// TIA Portal V19 export
FUNCTION_BLOCK "A0303_Manager_FB"   // FB14, LAD
// stored: MemoryReserve 100, SetENOAutomatically false
   VAR_INPUT
      AreaInterface : "AreaInterface";
      DataIn : Struct
         LsCheckPassaggio_Coda : Bool;   // FTC LETTURA STRATO DEPOSITATO TESTA
         LsCheckPassaggio_Testa : Bool;   // FTC LETTURA STRATO DEPOSITATO TESTA
         LsPezzoPosMax_Coda : Bool;
         LsPezzoPosMax_Testa : Bool;
         SemiAut_Pb : Bool;
      END_STRUCT;
      CIn : Struct
         PareggiatoreTesta : Struct
            Ax : "Positioning_DOL_Machine_COut";
         END_STRUCT;
         PareggiatoreCoda : Struct
            Ax : "Positioning_DOL_Machine_COut";
         END_STRUCT;
         Spalle : Struct
            Testa : Struct
               Ax : "Positioning_DOL_Machine_COut";
            END_STRUCT;
            Coda : Struct
               Ax : "Positioning_DOL_Machine_COut";
            END_STRUCT;
         END_STRUCT;
         Spintore : Struct
            Vrt : "ValveMachine_COut";
            Orz : "ValveMachine_COut";
         END_STRUCT;
         TraslazioneStrato : Struct
            Ax_Testa : "Positioning_EPOS_Machine_COut";
            Ax_Coda : "Positioning_EPOS_Machine_COut";
            Manip_Sostegno : "ValveMachine_COut";
            Manip_Pareggiatore : "ValveMachine_COut";
            SostegnoVrt : "ValveMachine_COut";
            IsMeasuring : Bool;
         END_STRUCT;
         Sollevamento : Struct
            Ax_Testa : "Positioning_DOL_Machine_COut";
            Ax_Coda : "Positioning_DOL_Machine_COut";
         END_STRUCT;
         Sostegno : Struct
            Testa : Struct
               Ax : "Positioning_DOL_Machine_COut";
               Paletto : Struct
                  CtrlSafe : Bool;
                  Standstill : Bool;
                  Rest_CheckNext : Bool;
                  Work_CheckNext : Bool;
                  Pos : Int;
                  RestPosition : Bool;
               END_STRUCT;
            END_STRUCT;
            Coda : Struct
               Ax : "Positioning_DOL_Machine_COut";
               Paletto : Struct
                  CtrlSafe : Bool;
                  Standstill : Bool;
                  Rest_CheckNext : Bool;
                  Work_CheckNext : Bool;
                  Pos : Int;
                  RestPosition : Bool;
               END_STRUCT;
            END_STRUCT;
         END_STRUCT;
         Navetta : Struct
            ReadyToRecive : Bool;
            OutOfWorkspace : Bool;
            InPosizioneDiDeposito : Bool;
            InPosizioneDiPrelievo : Bool;
            InPosizioneDiPrePrelievo : Bool;
            RequestDeposito : Bool;
            RequestPrelievo : Bool;
         END_STRUCT;
         ProdManager : "Prod_Beam_Ctrl";
      END_STRUCT;
   END_VAR
   VAR_OUTPUT
      MachineInterface : "MachineInterface";
      COut : Struct
         Spalla : Struct
            Testa : "Positioning_DOL_Machine_Manager";
            Coda : "Positioning_DOL_Machine_Manager";
         END_STRUCT;
         Spintore : Struct
            EnableStopDoorOpeningReq : Bool;
            EnableStopInPhase : Bool;
            EnableStopProgrammed : Bool;
            Control_ON : Bool;
            CanMoveFreely : Bool;
            Rest : Bool;
            Work : Bool;
         END_STRUCT;
         Trasporto : Struct
            EnableStopDoorOpeningReq : Bool;
            EnableStopInPhase : Bool;
            EnableStopProgrammed : Bool;
            Control_ON : Bool;
            CanMoveFreely : Bool;
            OP : Struct
               VAI_A_PRELIEVO : Bool;
               PRELIEVO : Bool;
               VAI_A_DEPOSITO : Bool;
               DEPOSITO : Bool;
            END_STRUCT;
         END_STRUCT;
         Sollevatore : Struct
            EnableStopDoorOpeningReq : Bool;
            EnableStopInPhase : Bool;
            EnableStopProgrammed : Bool;
            Control_ON : Bool;
            CanMoveFreely : Bool;
            TargetPosition : LReal;
            OP : Struct
               PRELIEVO : Bool;
               PRE_DEPOSITO : Bool;
               DEPOSITO : Bool;
            END_STRUCT;
         END_STRUCT;
         Sostegno : Struct
            Testa : Struct
               EnableStopDoorOpeningReq : Bool;
               EnableStopInPhase : Bool;
               EnableStopProgrammed : Bool;
               Control_ON : Bool;
               CanMoveFreely : Bool;
               Phase : Struct
                  VAI_A_LAVORO : Bool;
                  VAI_A_RIPOSO : Bool;
               END_STRUCT;
               Ax : Struct
                  Pos { ExternalVisible := 'False'; ExternalWritable := 'False'} : LReal;
               END_STRUCT;
               Paletti : Struct
                  PosPaletto : Int;
                  Pos1Collision : Bool;
                  Pos2Collision : Bool;
               END_STRUCT;
            END_STRUCT;
            Coda : Struct
               EnableStopDoorOpeningReq : Bool;
               EnableStopInPhase : Bool;
               EnableStopProgrammed : Bool;
               Control_ON : Bool;
               CanMoveFreely : Bool;
               Phase : Struct
                  VAI_A_LAVORO : Bool;
                  VAI_A_RIPOSO : Bool;
               END_STRUCT;
               Ax : Struct
                  Pos { ExternalVisible := 'False'; ExternalWritable := 'False'} : LReal;
               END_STRUCT;
               Paletti : Struct
                  PosPaletto : Int;
                  Pos1Collision : Bool;
                  Pos2Collision : Bool;
               END_STRUCT;
            END_STRUCT;
         END_STRUCT;
         Manipolatore : Struct
            ReadyToRecive : Bool;
         END_STRUCT;
      END_STRUCT;
   END_VAR
   VAR_IN_OUT
      Par : Struct
         Antiribaltamento : Struct
            Offset_Pos : LReal;
         END_STRUCT;
      END_STRUCT;
      Par_Trasporto : Struct
         PosPrelievo : LReal;
         PosDeposito : LReal;
         ToleranceWindow : LReal;
      END_STRUCT;
      Par_Sollevatore : Struct
         PosDeposito : LReal;
         OffsetPrelievo : LReal;
         ToleranceWindow : LReal;
      END_STRUCT;
      Par_SostegnoAntirib : Struct
         RestPosition : LReal;
         ToleranceWindow : LReal;
         PosTimeout : Time;
      END_STRUCT;
      Par_Spalla_Testa : Struct
         MinDistanzaConParegg : LReal;
         ToleranceWindow : LReal;
      END_STRUCT;
      Par_Spalla_Coda : Struct
         MinDistanzaConParegg : LReal;
         ToleranceWindow : LReal;
      END_STRUCT;
   END_VAR
   VAR
      Alarm : Struct
         TrkPassaggioPezzo : Bool;
         TrkPreparationAlreadyFull : Bool;
         TrkStackerAlreadyFull : Bool;
         PaccoOltreLimiteMax : Bool;
         STOP_FineTurno : Bool;
         STOP_End_Of_Proroduction : Bool;
         STOP_ControlloQualita : Bool;
         STOP_Inattività : Bool;
      END_STRUCT;
      Warning : Struct
         IsWaiting_NoPiecesBefore : Bool;
         IsWaiting_NoPiecesBefore_A01NotInCycle : Bool;
         IsWaiting_NoPiecesBefore_A02NotInCycle : Bool;
         IsWaiting_NoPiecesBefore_A03NotInCycle : Bool;
         IsWaiting_ShuttleUnload : Bool;
         IsWaiting_PezziDaRintegrare : Bool;
         STOP_End_Of_Proroduction : Bool;
         STOP_FineTurno : Bool;
         STOP_ControlloQualita : Bool;
         MissingCnd : Struct
            SollevatoreNotReadyToRecive : Bool;
         END_STRUCT;
      END_STRUCT;
      OP_CND : Struct
         Trasporto : Struct
            VaiAPrelievo : Array[0..15] of "OpCnd";
            Prelievo { S7_SetPoint := 'True'} : Array[0..15] of "OpCnd";
            VaiADeposito : Array[0..15] of "OpCnd";
            Deposito : Array[0..15] of "OpCnd";
         END_STRUCT;
      END_STRUCT;
      Ctrl : Struct
         Stop : Bool;
         Cycle : Struct
            Trasferimento : Struct
               VaiAPrelievo : Bool;   // CICLO - Vai a Posizione di prelievo
               Prelievo : Bool;   // CICLO - Prelievo
               VaiADeposito : Bool;   // CICLO - Vai a Posizione di deposito
               Deposito : Bool;   // CICLO - Deposito
            END_STRUCT;
            Sollevamento : Struct
               Prelievo : Bool;
               Deposito : Bool;
               PreDeposito : Bool;
            END_STRUCT;
            SostegnoAntirib_Testa : Struct
               VaiALavoro : Bool;
               VaiARiposo : Bool;
               CyclePos : LReal;
               PalettoPos : Int;
            END_STRUCT;
            SostegnoAntirib_Coda : Struct
               VaiALavoro : Bool;
               VaiARiposo : Bool;
               CyclePos : LReal;
               PalettoPos : Int;
            END_STRUCT;
         END_STRUCT;
         BTrk : Struct
            B3ToLayer1 : Bool;
            TransferToStacker : Bool;
         END_STRUCT;
         Spintore : Struct
            Vrt : Struct
               Rest : Bool;
               Work : Bool;
            END_STRUCT;
            Orz : Struct
               Rest : Bool;
               Work : Bool;
            END_STRUCT;
            Work : Bool;
            Rest : Bool;
         END_STRUCT;
         Spalle : Struct
            Testa : Struct
               MoveToPos : Bool;
               Pos : LReal;
            END_STRUCT;
            Coda : Struct
               MoveToPos : Bool;
               Pos : LReal;
            END_STRUCT;
         END_STRUCT;
         TraslazioneStrato : Struct
            Ax : Struct
               MovePrelievo : Bool;
               MoveDeposito : Bool;
               PosDeposito : LReal;
               PosPrelievo : LReal;
            END_STRUCT;
            SostegnoVrt : Struct
               Rest : Bool;
               Work : Bool;
            END_STRUCT;
            Manip_Sostegno : Struct
               Rest : Bool;
               Work : Bool;
            END_STRUCT;
            Manip_Pareggiatore : Struct
               Rest : Bool;
               Work : Bool;
            END_STRUCT;
         END_STRUCT;
      END_STRUCT;
      Sts : Struct
         AlarmsPresence : Bool;
         WarningsPresence : Bool;
         IsStandstill : Bool;
         SemiAut : Struct
            ON : Bool;
            PbMaterialFwd : Bool;
            Request : Bool;
         END_STRUCT;
         SpallaTesta : Struct
            InCyclePos : Bool;
         END_STRUCT;
         SpallaCoda : Struct
            InCyclePos : Bool;
         END_STRUCT;
         Sollevatore : Struct
            ReadyToRecive : Bool;
            InPrelievoPos : Bool;
            InPrePrelievoPos : Bool;
            InPosDeposito : Bool;
            InPosPreDeposito : Bool;
         END_STRUCT;
         Preparazione : Struct
            Completato : Bool;
         END_STRUCT;
         TraslazioneStrato : Struct
            InPosDeposito : Bool;
            InPosPrelievo : Bool;
            OutOfWorkspace : Bool;   // Fuori ingombro con sollevatore
            DropRequest : Bool;
         END_STRUCT;
         SostegnoTesta : Struct
            Ax : Struct
               InCyclePos : Bool;
               InRestPos : Bool;
            END_STRUCT;
            Paletto : Struct
               InCyclePos : Bool;
            END_STRUCT;
         END_STRUCT;
         SostegnoCoda : Struct
            Ax : Struct
               InCyclePos : Bool;
               InRestPos : Bool;
            END_STRUCT;
            Paletto : Struct
               InCyclePos : Bool;
            END_STRUCT;
         END_STRUCT;
         BTrk { ExternalAccessible := 'False'; ExternalVisible := 'False'; ExternalWritable := 'False'} : Struct
            ZonePreparationEmpty { S7_SetPoint := 'True'} : Bool;
            ZoneStackerEmpty : Bool;
            Actual_O_ID : DInt;
         END_STRUCT;
      END_STRUCT;
      AUX : Struct
         LsPosition1Coda_PE { ExternalAccessible := 'False'; ExternalVisible := 'False'; ExternalWritable := 'False'} : Bool;
         LsPosition1Coda_NE { ExternalAccessible := 'False'; ExternalVisible := 'False'; ExternalWritable := 'False'} : Bool;
         LsPosition1Testa_PE { ExternalAccessible := 'False'; ExternalVisible := 'False'; ExternalWritable := 'False'} : Bool;
         LsPosition1Testa_NE { ExternalAccessible := 'False'; ExternalVisible := 'False'; ExternalWritable := 'False'} : Bool;
         TrkToTransfer { ExternalAccessible := 'False'; ExternalVisible := 'False'; ExternalWritable := 'False'} : Bool;
         TrkToShuttle : Bool;
         SemiAut_Pb : Bool;
      END_STRUCT;
      TON_PassaggioPezzoAlarm : IEC_TIMER;
      TON_NoPiecesBefore : IEC_TIMER;
      TON_Stop { S7_SetPoint := 'True'} : IEC_TIMER;
      TON_StopPerInattivita { S7_SetPoint := 'True'} : IEC_TIMER;
      Attrezzamento : Struct
         Ready : Bool;
         FindNewID : Bool;
         RequestNewPosition : Bool;
         TargetSpalle : LReal;
         TargetSostegno : LReal;
         ID : DInt;
      END_STRUCT;
      CycleWithShortPiece : Bool;
      PE_Engaged_Coda : Bool;
      NE_Engaged_Coda : Bool;
      PE_Engaged_Testa : Bool;
      NE_Engaged_Testa : Bool;
      TON_CheckCompletato_Stacker : IEC_TIMER;
      TON_CheckCompletato_Preparation : IEC_TIMER;
   END_VAR
   VAR_TEMP
      PE : Struct
         LsPosition1_Coda : Bool;
         LsPosition1_Testa : Bool;
         TrkToTransfer : Bool;
         TrkToShuttle : Bool;
      END_STRUCT;
      NE : Struct
         LsPosition1_Coda : Bool;
         LsPosition1_Testa : Bool;
      END_STRUCT;
      BTrk_GetData : Struct   // BTrk letto dal MES
         indx : Int;   // Se trovato tra i TODO / ENDING / OUT questo è l'indice dove sono stati prelevati i dati
         Sts : Int;   // 0 = Non Trovato; 0 = ACT; 1 = TODO; 2=ENDING; 3 = OUT
         Item : "Prod_Item_small";
      END_STRUCT;
      BTrk_Absence : Bool;
      LayerTrk_Absence : Bool;
      O_ID_Precedenti : DInt;
      i : Int;
      EmptyNFound : Int;
      ShiftN : Int;
      TargetPrePositionSollevatore : LReal;
      TargetPositionSollevatore_Temp : LReal;
      TargetPositionSollevatore : LReal;
      TargetPreDepositoSollevatore : LReal;
      SollevatoreCodaInPrelievoPos : Bool;
      SollevatoreTestaInPrelievoPos : Bool;
      SollevatoreCodaInPrePrelievoPos : Bool;
      SollevatoreTestaInPrePrelievoPos : Bool;
      SollevatoreCodaInPosDeposito : Bool;
      SollevatoreTestaInPosDeposito : Bool;
      SollevatoreTestaInPosPreDeposito : Bool;
      SollevatoreCodaInPosPreDeposito : Bool;
      TrasportoTestaInPosDeposito : Bool;
      TrasportoTestaInPosPrelievo : Bool;
      TrasportoCodaInPosDeposito : Bool;
      TrasportoCodaInPosPrelievo : Bool;
      ShiftArrayOk : Int;
      TrkToStackerOk : Int;
      PieceToCheck_Presence : Bool;
      O_ID_Temp : DInt;
      ConteggioPezzi_Preparation : Int;
      ConteggioPezzi_Stacker : Int;
      ConteggioPezzi_Transfert : Int;
      MaxBeamsXLayer : Int;
      MaxLayer : Int;
   END_VAR
   VAR CONSTANT
      TrasportoOutOfWorkspace : LReal := -215.0;
   END_VAR
   VAR_TEMP   // added for the SCL form of the ladder/FBD networks
      _w1 : Bool;
      _w2 : Bool;
      _w3 : Bool;
      _w4 : Bool;
      _w5 : Bool;
   END_VAR
BEGIN

REGION Network 1 (SCL): Reset Alarms
   IF #AreaInterface.RstAlarms THEN
       #Alarm.TrkPassaggioPezzo := FALSE;
       #Alarm.TrkPreparationAlreadyFull := FALSE;
       #Alarm.TrkStackerAlreadyFull := FALSE;
       #Alarm.PaccoOltreLimiteMax := FALSE;
       #Alarm.STOP_End_Of_Proroduction := FALSE;
       #Alarm.STOP_FineTurno := FALSE;
       #Alarm.STOP_ControlloQualita := FALSE;
   END_IF;
END_REGION

REGION Network 2: Fronti Sensori
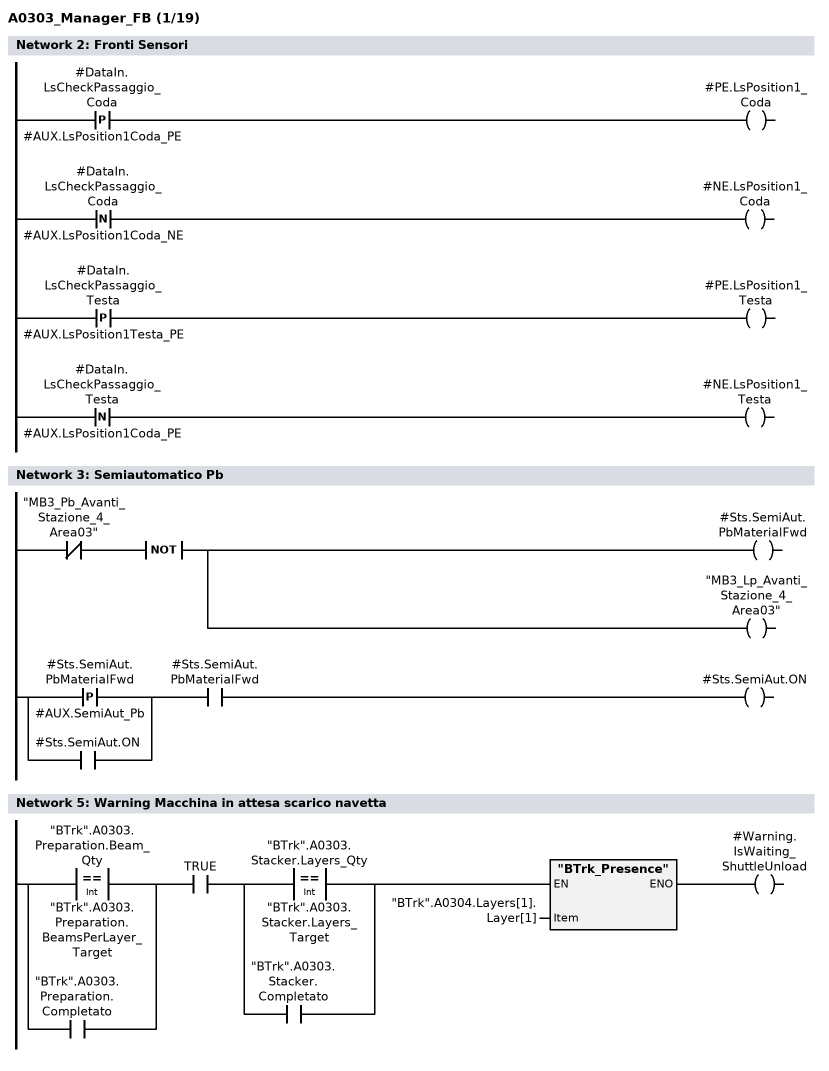
   RUNG wire#powerrail
      P_Contact(operand := #DataIn.LsCheckPassaggio_Coda, bit := #AUX.LsPosition1Coda_PE)
      Coil( #PE.LsPosition1_Coda )
   END_RUNG
   RUNG wire#powerrail
      N_Contact(operand := #DataIn.LsCheckPassaggio_Coda, bit := #AUX.LsPosition1Coda_NE)
      Coil( #NE.LsPosition1_Coda )
   END_RUNG
   RUNG wire#powerrail
      P_Contact(operand := #DataIn.LsCheckPassaggio_Testa, bit := #AUX.LsPosition1Testa_PE)
      Coil( #PE.LsPosition1_Testa )
   END_RUNG
   RUNG wire#powerrail
      N_Contact(operand := #DataIn.LsCheckPassaggio_Testa, bit := #AUX.LsPosition1Coda_PE)
      Coil( #NE.LsPosition1_Testa )
   END_RUNG
   // the same network as SCL:
   #_w1 := #DataIn.LsCheckPassaggio_Coda AND NOT #AUX.LsPosition1Coda_PE;   // rising edge of #DataIn.LsCheckPassaggio_Coda
   #AUX.LsPosition1Coda_PE := #DataIn.LsCheckPassaggio_Coda;
   #PE.LsPosition1_Coda := #_w1;
   #_w2 := NOT #DataIn.LsCheckPassaggio_Coda AND #AUX.LsPosition1Coda_NE;   // falling edge of #DataIn.LsCheckPassaggio_Coda
   #AUX.LsPosition1Coda_NE := #DataIn.LsCheckPassaggio_Coda;
   #NE.LsPosition1_Coda := #_w2;
   #_w3 := #DataIn.LsCheckPassaggio_Testa AND NOT #AUX.LsPosition1Testa_PE;   // rising edge of #DataIn.LsCheckPassaggio_Testa
   #AUX.LsPosition1Testa_PE := #DataIn.LsCheckPassaggio_Testa;
   #PE.LsPosition1_Testa := #_w3;
   #_w4 := NOT #DataIn.LsCheckPassaggio_Testa AND #AUX.LsPosition1Coda_PE;   // falling edge of #DataIn.LsCheckPassaggio_Testa
   #AUX.LsPosition1Coda_PE := #DataIn.LsCheckPassaggio_Testa;
   #NE.LsPosition1_Testa := #_w4;
END_REGION

REGION Network 3: Semiautomatico Pb
   RUNG wire#powerrail
      I_Contact( "MB3_Pb_Avanti_Stazione_4_Area03" )
      Not()
      wire#w1
      Coil( #Sts.SemiAut.PbMaterialFwd )
   END_RUNG
   RUNG wire#w1
      Coil( "MB3_Lp_Avanti_Stazione_4_Area03" )
   END_RUNG
   RUNG wire#powerrail
      P_Contact(operand := #Sts.SemiAut.PbMaterialFwd, bit := #AUX.SemiAut_Pb)
      wire#w2
      Contact( #Sts.SemiAut.PbMaterialFwd )
      Coil( #Sts.SemiAut.ON )
   END_RUNG
   RUNG wire#powerrail
      Contact( #Sts.SemiAut.ON )
   END_RUNG wire#w2
   // the same network as SCL:
   #Sts.SemiAut.PbMaterialFwd := NOT (NOT "MB3_Pb_Avanti_Stazione_4_Area03");
   "MB3_Lp_Avanti_Stazione_4_Area03" := NOT (NOT "MB3_Pb_Avanti_Stazione_4_Area03");
   #_w1 := #Sts.SemiAut.PbMaterialFwd AND NOT #AUX.SemiAut_Pb;   // rising edge of #Sts.SemiAut.PbMaterialFwd
   #AUX.SemiAut_Pb := #Sts.SemiAut.PbMaterialFwd;
   #Sts.SemiAut.ON := (#_w1 OR #Sts.SemiAut.ON) AND #Sts.SemiAut.PbMaterialFwd;
END_REGION

REGION Network 5: Warning Macchina in attesa scarico navetta
   RUNG wire#powerrail
      { S7_Templates := "SrcType := Int" } EQ_Contact(in1 := "BTrk".A0303.Preparation.Beam_Qty, in2 := "BTrk".A0303.Preparation.BeamsPerLayer_Target)
      wire#w1
      Contact( TRUE )
      wire#w2
      { S7_Templates := "SrcType := Int" } EQ_Contact(in1 := "BTrk".A0303.Stacker.Layers_Qty, in2 := "BTrk".A0303.Stacker.Layers_Target)
      wire#w3
      "BTrk_Presence"(Item := "BTrk".A0304.Layers[1].Layer[1])
      Coil( #Warning.IsWaiting_ShuttleUnload )
   END_RUNG
   RUNG wire#powerrail
      Contact( "BTrk".A0303.Preparation.Completato )
   END_RUNG wire#w1
   RUNG wire#w2
      Contact( "BTrk".A0303.Stacker.Completato )
   END_RUNG wire#w3
   // the same network as SCL:
   "BTrk_Presence"(EN := (("BTrk".A0303.Preparation.Beam_Qty = "BTrk".A0303.Preparation.BeamsPerLayer_Target) OR "BTrk".A0303.Preparation.Completato) AND TRUE AND (("BTrk".A0303.Stacker.Layers_Qty = "BTrk".A0303.Stacker.Layers_Target) OR "BTrk".A0303.Stacker.Completato),
                   Item := "BTrk".A0304.Layers[1].Layer[1],
                   ENO => #_w1);
   #Warning.IsWaiting_ShuttleUnload := #_w1;
END_REGION

REGION Network 6: Warning Macchina in attesa nessun pezzo in arrivo
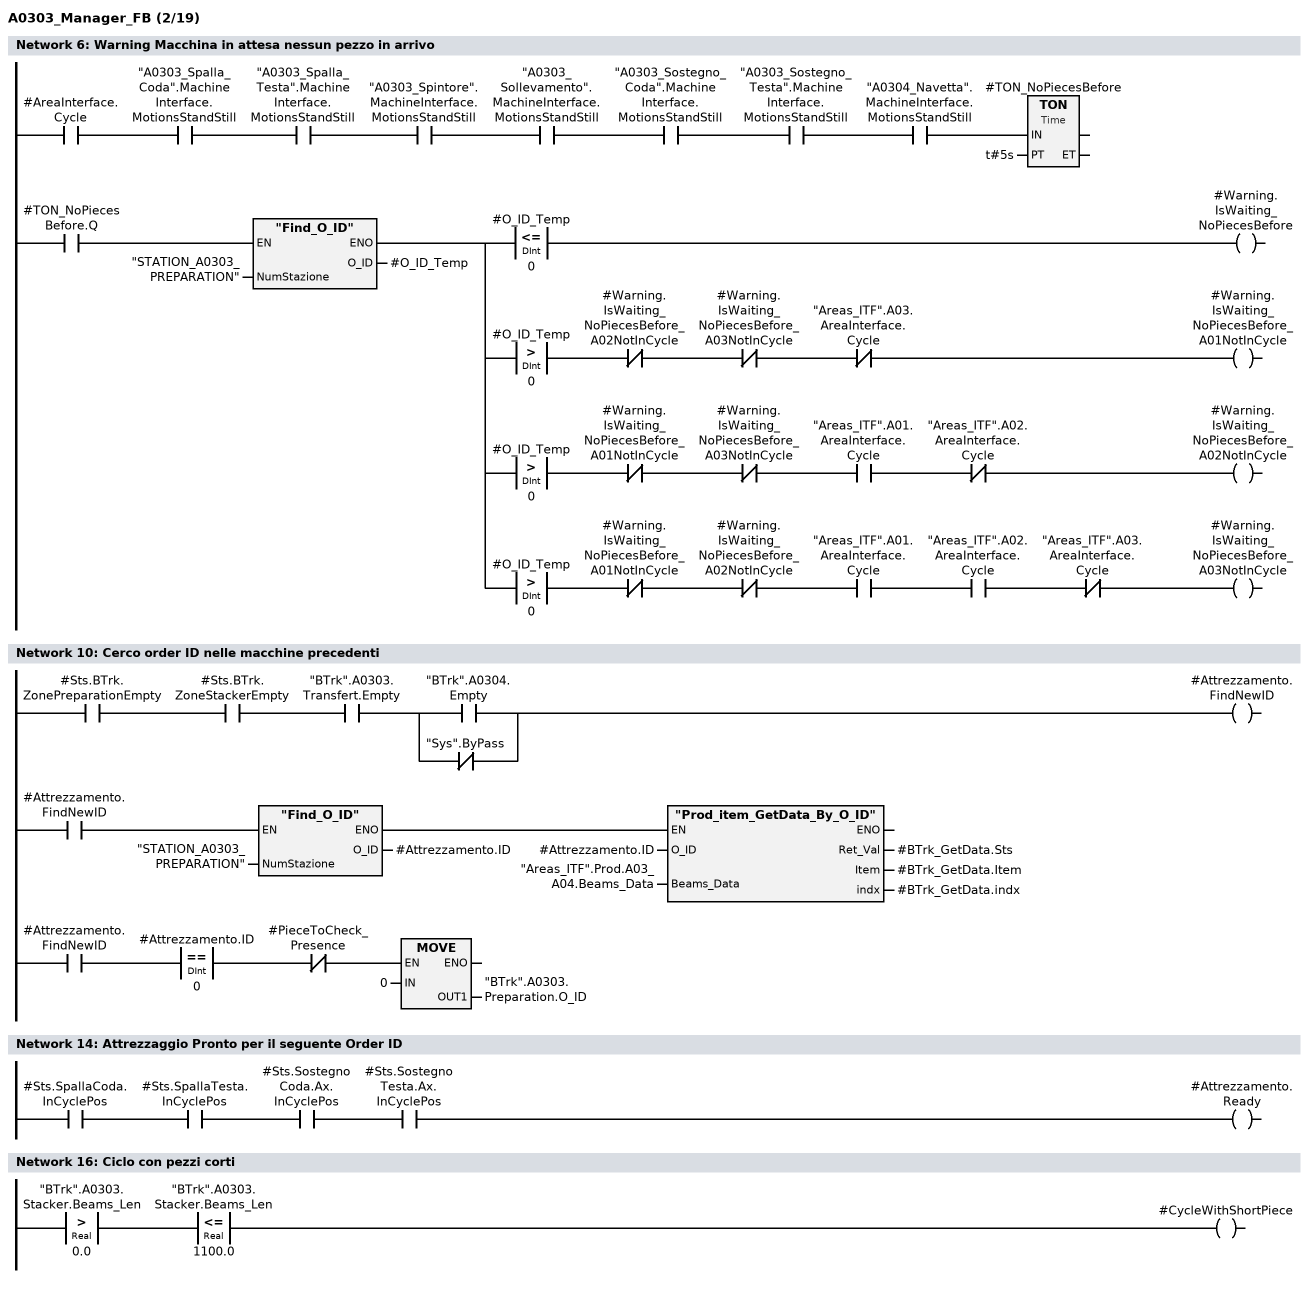
   RUNG wire#powerrail
      Contact( #AreaInterface.Cycle )
      Contact( "A0303_Spalla_Coda".MachineInterface.MotionsStandStill )
      Contact( "A0303_Spalla_Testa".MachineInterface.MotionsStandStill )
      Contact( "A0303_Spintore".MachineInterface.MotionsStandStill )
      Contact( "A0303_Sollevamento".MachineInterface.MotionsStandStill )
      Contact( "A0303_Sostegno_Coda".MachineInterface.MotionsStandStill )
      Contact( "A0303_Sostegno_Testa".MachineInterface.MotionsStandStill )
      Contact( "A0304_Navetta".MachineInterface.MotionsStandStill )
      { S7_Templates := "time_type := Time" } #TON_NoPiecesBefore.TON(pt := t#5s, et =>)
   END_RUNG
   RUNG wire#powerrail
      Contact( #TON_NoPiecesBefore.Q )
      "Find_O_ID"(NumStazione := "STATION_A0303_PREPARATION", O_ID => #O_ID_Temp)
      wire#w1
      { S7_Templates := "SrcType := DInt" } LE_Contact(in1 := #O_ID_Temp, in2 := 0)
      Coil( #Warning.IsWaiting_NoPiecesBefore )
   END_RUNG
   RUNG wire#w1
      { S7_Templates := "SrcType := DInt" } GT_Contact(in1 := #O_ID_Temp, in2 := 0)
      I_Contact( #Warning.IsWaiting_NoPiecesBefore_A02NotInCycle )
      I_Contact( #Warning.IsWaiting_NoPiecesBefore_A03NotInCycle )
      I_Contact( "Areas_ITF".A03.AreaInterface.Cycle )
      Coil( #Warning.IsWaiting_NoPiecesBefore_A01NotInCycle )
   END_RUNG
   RUNG wire#w1
      { S7_Templates := "SrcType := DInt" } GT_Contact(in1 := #O_ID_Temp, in2 := 0)
      I_Contact( #Warning.IsWaiting_NoPiecesBefore_A01NotInCycle )
      I_Contact( #Warning.IsWaiting_NoPiecesBefore_A03NotInCycle )
      Contact( "Areas_ITF".A01.AreaInterface.Cycle )
      I_Contact( "Areas_ITF".A02.AreaInterface.Cycle )
      Coil( #Warning.IsWaiting_NoPiecesBefore_A02NotInCycle )
   END_RUNG
   RUNG wire#w1
      { S7_Templates := "SrcType := DInt" } GT_Contact(in1 := #O_ID_Temp, in2 := 0)
      I_Contact( #Warning.IsWaiting_NoPiecesBefore_A01NotInCycle )
      I_Contact( #Warning.IsWaiting_NoPiecesBefore_A02NotInCycle )
      Contact( "Areas_ITF".A01.AreaInterface.Cycle )
      Contact( "Areas_ITF".A02.AreaInterface.Cycle )
      I_Contact( "Areas_ITF".A03.AreaInterface.Cycle )
      Coil( #Warning.IsWaiting_NoPiecesBefore_A03NotInCycle )
   END_RUNG
   // the same network as SCL:
   #TON_NoPiecesBefore.TON(IN := #AreaInterface.Cycle AND "A0303_Spalla_Coda".MachineInterface.MotionsStandStill AND "A0303_Spalla_Testa".MachineInterface.MotionsStandStill AND "A0303_Spintore".MachineInterface.MotionsStandStill AND "A0303_Sollevamento".MachineInterface.MotionsStandStill AND "A0303_Sostegno_Coda".MachineInterface.MotionsStandStill AND "A0303_Sostegno_Testa".MachineInterface.MotionsStandStill AND "A0304_Navetta".MachineInterface.MotionsStandStill,
                           PT := t#5s);
   "Find_O_ID"(EN := #TON_NoPiecesBefore.Q,
               NumStazione := "STATION_A0303_PREPARATION",
               O_ID => #O_ID_Temp,
               ENO => #_w1);
   #Warning.IsWaiting_NoPiecesBefore := #_w1 AND (#O_ID_Temp <= 0);
   #Warning.IsWaiting_NoPiecesBefore_A01NotInCycle := #_w1 AND (#O_ID_Temp > 0) AND NOT #Warning.IsWaiting_NoPiecesBefore_A02NotInCycle AND NOT #Warning.IsWaiting_NoPiecesBefore_A03NotInCycle AND NOT "Areas_ITF".A03.AreaInterface.Cycle;
   #Warning.IsWaiting_NoPiecesBefore_A02NotInCycle := #_w1 AND (#O_ID_Temp > 0) AND NOT #Warning.IsWaiting_NoPiecesBefore_A01NotInCycle AND NOT #Warning.IsWaiting_NoPiecesBefore_A03NotInCycle AND "Areas_ITF".A01.AreaInterface.Cycle AND NOT "Areas_ITF".A02.AreaInterface.Cycle;
   #Warning.IsWaiting_NoPiecesBefore_A03NotInCycle := #_w1 AND (#O_ID_Temp > 0) AND NOT #Warning.IsWaiting_NoPiecesBefore_A01NotInCycle AND NOT #Warning.IsWaiting_NoPiecesBefore_A02NotInCycle AND "Areas_ITF".A01.AreaInterface.Cycle AND "Areas_ITF".A02.AreaInterface.Cycle AND NOT "Areas_ITF".A03.AreaInterface.Cycle;
END_REGION

REGION Network 7: <<<<<<<<<<<<<<<<<<<<<<<<<<<<<<<<< ZONA 303 ATTREZZAGGIO >>>>>>>>>>>>>>>>>>>>>>>>>>>>>>>>>>>>
END_REGION

REGION Network 8 (SCL): Zona Vuota
   //CONTROLLO CHE CI SIANO LE CONDIZIONI PER MUOVERSI (TRK EMPTY)
   //
   FOR #i := 1 TO "BTRK_A0303_ITEMS" DO
       IF "BTrk".A0303.Preparation.B.B_ID = 0 THEN
           #BTrk_Absence := TRUE;
       ELSE
           #BTrk_Absence := FALSE;
           EXIT;
       END_IF;
   END_FOR;

   FOR #i := 1 TO "BTRK_LAYER_ITEMS" DO
       IF "BTrk".A0303.Preparation.Layer[#i].B_ID = 0 THEN
           #LayerTrk_Absence := TRUE;
       ELSE
           #LayerTrk_Absence := FALSE;
           EXIT;
       END_IF;
   END_FOR;


   #Sts.BTrk.ZonePreparationEmpty := #BTrk_Absence AND #LayerTrk_Absence AND NOT #DataIn.LsCheckPassaggio_Coda;
   #Sts.BTrk.ZoneStackerEmpty := "BTrk".A0303.Stacker.Empty;
END_REGION

REGION Network 9 (SCL): A03_EXIT_TOCHECK controllo che accumulo non abbia pezzi da controllare o rintegrati
   #PieceToCheck_Presence:="PieceToCheck_Presence"(Trk_B:="BTrk".A03_EXIT_TOCHECK.B) ;
END_REGION

REGION Network 10: Cerco order ID nelle macchine precedenti
   RUNG wire#powerrail
      Contact( #Sts.BTrk.ZonePreparationEmpty )
      Contact( #Sts.BTrk.ZoneStackerEmpty )
      Contact( "BTrk".A0303.Transfert.Empty )
      wire#w1
      Contact( "BTrk".A0304.Empty )
      wire#w2
      Coil( #Attrezzamento.FindNewID )
   END_RUNG
   RUNG wire#w1
      I_Contact( "Sys".ByPass )
   END_RUNG wire#w2
   RUNG wire#powerrail
      Contact( #Attrezzamento.FindNewID )
      "Find_O_ID"(NumStazione := "STATION_A0303_PREPARATION", O_ID => #Attrezzamento.ID)
      "Prod_item_GetData_By_O_ID"(O_ID := #Attrezzamento.ID, Beams_Data := "Areas_ITF".Prod.A03_A04.Beams_Data, Ret_Val => #BTrk_GetData.Sts, Item => #BTrk_GetData.Item, indx => #BTrk_GetData.indx)
   END_RUNG
   RUNG wire#powerrail
      Contact( #Attrezzamento.FindNewID )
      { S7_Templates := "SrcType := DInt" } EQ_Contact(in1 := #Attrezzamento.ID, in2 := 0)
      I_Contact( #PieceToCheck_Presence )
      Move(in := 0, out1 => "BTrk".A0303.Preparation.O_ID)
   END_RUNG
   // the same network as SCL:
   #Attrezzamento.FindNewID := #Sts.BTrk.ZonePreparationEmpty AND #Sts.BTrk.ZoneStackerEmpty AND "BTrk".A0303.Transfert.Empty AND ("BTrk".A0304.Empty OR NOT "Sys".ByPass);
   "Find_O_ID"(EN := #Attrezzamento.FindNewID,
               NumStazione := "STATION_A0303_PREPARATION",
               O_ID => #Attrezzamento.ID,
               ENO => #_w1);
   IF #_w1 THEN
       #BTrk_GetData.Sts := "Prod_item_GetData_By_O_ID"(O_ID := #Attrezzamento.ID,
                               Beams_Data := "Areas_ITF".Prod.A03_A04.Beams_Data,
                               Item => #BTrk_GetData.Item,
                               indx => #BTrk_GetData.indx);
   END_IF;
   IF #Attrezzamento.FindNewID AND (#Attrezzamento.ID = 0) AND NOT #PieceToCheck_Presence THEN
       "BTrk".A0303.Preparation.O_ID := 0;
   END_IF;
END_REGION

REGION Network 11 (SCL): Numero Max Beams per Layer / Numero Max Layer
   CASE REAL_TO_INT(IN:="BTrk".A0303.Preparation.Beam_H_B )OF

       0:
           ;
       60:
           #MaxBeamsXLayer := "STACK_BEAMS_PER_LAYER_QTY_MAX_C060";
           #MaxLayer := "STACK_LAYERS_QTY_MAX_C060";
       70:
           #MaxBeamsXLayer := "STACK_BEAMS_PER_LAYER_QTY_MAX_C070";
           #MaxLayer := "STACK_LAYERS_QTY_MAX_C070";
       80:
           #MaxBeamsXLayer := "STACK_BEAMS_PER_LAYER_QTY_MAX_C080";
           #MaxLayer := "STACK_LAYERS_QTY_MAX_C080";
       90:
           #MaxBeamsXLayer := "STACK_BEAMS_PER_LAYER_QTY_MAX_C090";
           #MaxLayer := "STACK_LAYERS_QTY_MAX_C090";
       100:
           #MaxBeamsXLayer := "STACK_BEAMS_PER_LAYER_QTY_MAX_C100";
           #MaxLayer := "STACK_LAYERS_QTY_MAX_C100";
       110:
           #MaxBeamsXLayer := "STACK_BEAMS_PER_LAYER_QTY_MAX_C110";
           #MaxLayer := "STACK_LAYERS_QTY_MAX_C110";
       120:
           #MaxBeamsXLayer := "STACK_BEAMS_PER_LAYER_QTY_MAX_C120";
           #MaxLayer := "STACK_LAYERS_QTY_MAX_C120";
       130:
           #MaxBeamsXLayer := "STACK_BEAMS_PER_LAYER_QTY_MAX_C130";
           #MaxLayer := "STACK_LAYERS_QTY_MAX_C130";
       140:
           #MaxBeamsXLayer := "STACK_BEAMS_PER_LAYER_QTY_MAX_C140";
           #MaxLayer := "STACK_LAYERS_QTY_MAX_C140";
       150:
           #MaxBeamsXLayer := "STACK_BEAMS_PER_LAYER_QTY_MAX_C150";
           #MaxLayer := "STACK_LAYERS_QTY_MAX_C150";
       180:
           #MaxBeamsXLayer := "STACK_BEAMS_PER_LAYER_QTY_MAX_C180";
           #MaxLayer := "STACK_LAYERS_QTY_MAX_C180";
       200:
           #MaxBeamsXLayer := "STACK_BEAMS_PER_LAYER_QTY_MAX_C200";
           #MaxLayer := "STACK_LAYERS_QTY_MAX_C200";





   END_CASE;
END_REGION

REGION Network 12 (SCL): Compilo i dati del btrk in base all'order ID in arrivo
   IF #BTrk_GetData.Sts >= 0 AND #BTrk_GetData.Item.Beam_Code = 1 THEN

       "BTrk".A0303.Preparation.O_ID :="BTrk".A0303.Transfert.O_ID:="BTrk".A0303.Stacker.O_ID:="BTrk".A0304.O_ID:=#Attrezzamento.ID;
       "BTrk".A0303.Preparation.Beam_Len:= "BTrk".A0303.Transfert.Beams_Len := "BTrk".A0303.Stacker.Beams_Len := "BTrk".A0304.Beams_Len := #BTrk_GetData.Item.Beams_Len;
       "BTrk".A0303.Preparation.BeamsPerLayer_Target := "BTrk".A0303.Transfert.BeamsPerLayer_Target := "BTrk".A0303.Stacker.BeamsPerLayer_Target := "BTrk".A0304.BeamsPerLayer_Target := MIN(IN1 := #BTrk_GetData.Item.PackLayout_BeamsPerLayer, IN2 := #MaxBeamsXLayer);
       "BTrk".A0303.Preparation.Layers_Target := "BTrk".A0303.Transfert.Layers_Target := "BTrk".A0303.Stacker.Layers_Target := "BTrk".A0304.Layers_Target := MIN(IN1 := #BTrk_GetData.Item.PackLayout_Layers_Qty, IN2 := #MaxLayer);
       "BTrk".A0303.Preparation.Beam_H_B := "BTrk".A0303.Transfert.Beams_H_B := "BTrk".A0303.Stacker.Beams_H_B := "BTrk".A0304.Beams_H_B := #BTrk_GetData.Item.Beams_H_B;
       "BTrk".A0303.Preparation.Beam_W_A := "BTrk".A0303.Transfert.Beams_W_A := "BTrk".A0303.Stacker.Beams_W_A := "BTrk".A0304.Beams_W_A := #BTrk_GetData.Item.Beams_W_A;


   ELSE
       IF "BTrk".A0303.Preparation.O_ID <= 0 THEN

           "BTrk".A0303.Preparation.O_ID := "BTrk".A0303.Transfert.O_ID := "BTrk".A0303.Stacker.O_ID := "BTrk".A0304.O_ID := -1;
           "BTrk".A0303.Preparation.Beam_Len := "BTrk".A0303.Transfert.Beams_Len := "BTrk".A0303.Stacker.Beams_Len := "BTrk".A0304.Beams_Len := -1;
           "BTrk".A0303.Preparation.BeamsPerLayer_Target := "BTrk".A0303.Transfert.BeamsPerLayer_Target := "BTrk".A0303.Stacker.BeamsPerLayer_Target := "BTrk".A0304.BeamsPerLayer_Target := -1;
           "BTrk".A0303.Preparation.Layers_Target := "BTrk".A0303.Transfert.Layers_Target := "BTrk".A0303.Stacker.Layers_Target := "BTrk".A0304.Layers_Target := -1;
           "BTrk".A0303.Preparation.Beam_H_B := "BTrk".A0303.Transfert.Beams_H_B := "BTrk".A0303.Stacker.Beams_H_B := "BTrk".A0304.Beams_H_B := -1;
           "BTrk".A0303.Preparation.Beam_W_A := "BTrk".A0303.Transfert.Beams_W_A := "BTrk".A0303.Stacker.Beams_W_A := "BTrk".A0304.Beams_W_A := -1;

       END_IF;

       ;
   END_IF;
END_REGION

REGION Network 13 (SCL): Richiesta nuovo posizionamento x cambio Order ID
   #Attrezzamento.RequestNewPosition := ("BTrk".A0303.Preparation.O_ID <> -1)
                                       AND (#BTrk_GetData.Sts >= 0)
                                       AND (#BTrk_GetData.Item.Beam_Code = 1)
                                       AND #Attrezzamento.FindNewID
                                       AND NOT #Attrezzamento.Ready
                                       AND NOT #PieceToCheck_Presence;
END_REGION

REGION Network 14: Attrezzaggio Pronto per il seguente Order ID
   RUNG wire#powerrail
      Contact( #Sts.SpallaCoda.InCyclePos )
      Contact( #Sts.SpallaTesta.InCyclePos )
      Contact( #Sts.SostegnoCoda.Ax.InCyclePos )
      Contact( #Sts.SostegnoTesta.Ax.InCyclePos )
      Coil( #Attrezzamento.Ready )
   END_RUNG
   // the same network as SCL:
   #Attrezzamento.Ready := #Sts.SpallaCoda.InCyclePos AND #Sts.SpallaTesta.InCyclePos AND #Sts.SostegnoCoda.Ax.InCyclePos AND #Sts.SostegnoTesta.Ax.InCyclePos;
END_REGION

REGION Network 15 (SCL): Target Posizionamento Spalle e Sostegno
   IF "BTrk".A0303.Preparation.Beam_Len > 0 THEN
       //Posiziono le spalle in base alla lunghezza dei pezzi
       #Attrezzamento.TargetSpalle := ("BTrk".A0303.Preparation.Beam_Len / 2.0);

       //Posiziono il sostegno in base alla larghezza del pezzo e il numero di pezzi per riga
       #Attrezzamento.TargetSostegno := ("BTrk".A0303.Preparation.Beam_H_B* "BTrk".A0303.Preparation.BeamsPerLayer_Target)+#Par.Antiribaltamento.Offset_Pos;

   ELSE
       #Attrezzamento.TargetSpalle := -1;

       #Attrezzamento.TargetSostegno := -1;

   END_IF;
END_REGION

REGION Network 16: Ciclo con pezzi corti
   RUNG wire#powerrail
      { S7_Templates := "SrcType := Real" } GT_Contact(in1 := "BTrk".A0303.Stacker.Beams_Len, in2 := 0.0)
      { S7_Templates := "SrcType := Real" } LE_Contact(in1 := "BTrk".A0303.Stacker.Beams_Len, in2 := 1100.0)
      Coil( #CycleWithShortPiece )
   END_RUNG
   // the same network as SCL:
   #CycleWithShortPiece := ("BTrk".A0303.Stacker.Beams_Len > 0.0) AND ("BTrk".A0303.Stacker.Beams_Len <= 1100.0);
END_REGION

REGION Network 17 (SCL): Pacco Completato su preparation anche se non completo perche finiti i pezzi dello stesso Order ID
   IF NOT "BTrk".A0303.Preparation.Empty OR NOT "Sys".ByPass THEN

      // Cerco se nelle stazioni precedenti ci sono pezzi con lo stesso Order Id  

       "Find_O_ID"(NumStazione:="STATION_A0303_PREPARATION",O_ID=>#O_ID_Precedenti);
       #TON_CheckCompletato_Preparation.TON(IN := ((#O_ID_Precedenti <> "BTrk".A0303.Preparation.O_ID) (*AND ("Areas_ITF".Prod.A03_A04.Beams_Data.O_ACT.O_ID <> "BTrk".A0303.Preparation.O_ID)*)),
                                            PT := T#10s);


       IF #TON_CheckCompletato_Preparation.Q THEN

           "BTrk".A0303.Preparation.Completato := NOT #PieceToCheck_Presence;

        END_IF;


    END_IF;
END_REGION

REGION Network 18 (SCL): Pacco Completato su Stacker anche se non completo perche finiti i pezzi dello stesso Order ID
   IF NOT "BTrk".A0303.Stacker.Empty THEN

      // Cerco se nelle stazioni precedenti ci sono pezzi con lo stesso Order Id  

       "Find_O_ID"(NumStazione:="STATION_A0303_STACKER",O_ID=>#O_ID_Precedenti);
       #TON_CheckCompletato_Stacker.TON(IN:=((((#O_ID_Precedenti <> "BTrk".A0303.Stacker.O_ID)) AND ("Areas_ITF".Prod.A03_A04.Beams_Data.O_ACT.O_ID <> "BTrk".A0303.Stacker.O_ID )) AND "BTrk".A0303.Transfert.Empty AND "BTrk".A0303.Preparation.Empty),PT := T#10S);

       IF #TON_CheckCompletato_Stacker.Q THEN

           "BTrk".A0303.Stacker.Completato := NOT #PieceToCheck_Presence;

        END_IF;


    END_IF;
END_REGION

REGION Network 19: <<<<<<<<<<<<<<<<<<<<<<<<<<<<<<<<<<< PREPARAZIONE STRATO >>>>>>>>>>>>>>>>>>>>>>>>>>>>>>>>>>>>>>
END_REGION

REGION Network 20: <<< POSIZIONAMENTO SPALLE >>>
END_REGION

REGION Network 21: Ax Spalla in posizione
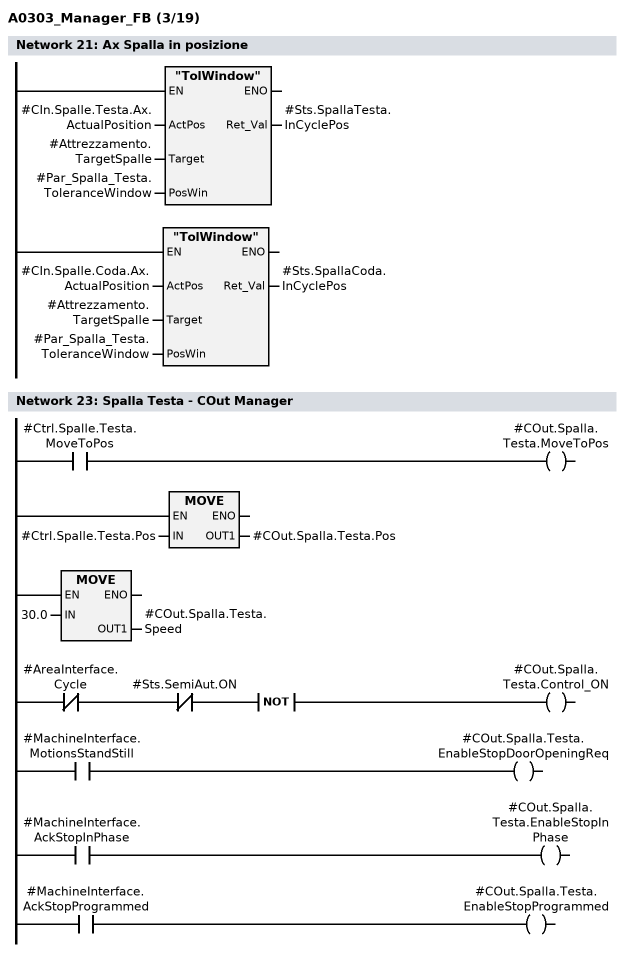
   RUNG wire#powerrail
      "TolWindow"(ActPos := #CIn.Spalle.Testa.Ax.ActualPosition, Target := #Attrezzamento.TargetSpalle, PosWin := #Par_Spalla_Testa.ToleranceWindow, Ret_Val => #Sts.SpallaTesta.InCyclePos)
   END_RUNG
   RUNG wire#powerrail
      "TolWindow"(ActPos := #CIn.Spalle.Coda.Ax.ActualPosition, Target := #Attrezzamento.TargetSpalle, PosWin := #Par_Spalla_Testa.ToleranceWindow, Ret_Val => #Sts.SpallaCoda.InCyclePos)
   END_RUNG
   // the same network as SCL:
   #Sts.SpallaTesta.InCyclePos := "TolWindow"(ActPos := #CIn.Spalle.Testa.Ax.ActualPosition,
                           Target := #Attrezzamento.TargetSpalle,
                           PosWin := #Par_Spalla_Testa.ToleranceWindow);
   #Sts.SpallaCoda.InCyclePos := "TolWindow"(ActPos := #CIn.Spalle.Coda.Ax.ActualPosition,
                           Target := #Attrezzamento.TargetSpalle,
                           PosWin := #Par_Spalla_Testa.ToleranceWindow);
END_REGION

REGION Network 22 (SCL): Comando Posizionamento Spalle
   //Spalla di TESTA


   IF (NOT #Sts.SpallaTesta.InCyclePos  AND (#Attrezzamento.TargetSpalle <> -1 )) AND #Sts.SostegnoTesta.Ax.InRestPos THEN
       #Ctrl.Spalle.Testa.Pos := #Attrezzamento.TargetSpalle;
       #Ctrl.Spalle.Testa.MoveToPos := #Attrezzamento.RequestNewPosition;
   ELSE
       #Ctrl.Spalle.Testa.MoveToPos := FALSE;
   END_IF;


   //Spalla di CODA
   //


   IF (NOT #Sts.SpallaCoda.InCyclePos AND ( #Attrezzamento.TargetSpalle <> -1)) AND #Sts.SostegnoCoda.Ax.InRestPos THEN
       #Ctrl.Spalle.Coda.Pos := #Attrezzamento.TargetSpalle;
       #Ctrl.Spalle.Coda.MoveToPos := #Attrezzamento.RequestNewPosition;

   ELSE
       #Ctrl.Spalle.Coda.MoveToPos := FALSE;
   END_IF;
END_REGION

REGION Network 23: Spalla Testa - COut Manager
   RUNG wire#powerrail
      Contact( #Ctrl.Spalle.Testa.MoveToPos )
      Coil( #COut.Spalla.Testa.MoveToPos )
   END_RUNG
   RUNG wire#powerrail
      Move(in := #Ctrl.Spalle.Testa.Pos, out1 => #COut.Spalla.Testa.Pos)
   END_RUNG
   RUNG wire#powerrail
      Move(in := 30.0, out1 => #COut.Spalla.Testa.Speed)
   END_RUNG
   RUNG wire#powerrail
      I_Contact( #AreaInterface.Cycle )
      I_Contact( #Sts.SemiAut.ON )
      Not()
      Coil( #COut.Spalla.Testa.Control_ON )
   END_RUNG
   RUNG wire#powerrail
      Contact( #MachineInterface.MotionsStandStill )
      Coil( #COut.Spalla.Testa.EnableStopDoorOpeningReq )
   END_RUNG
   RUNG wire#powerrail
      Contact( #MachineInterface.AckStopInPhase )
      Coil( #COut.Spalla.Testa.EnableStopInPhase )
   END_RUNG
   RUNG wire#powerrail
      Contact( #MachineInterface.AckStopProgrammed )
      Coil( #COut.Spalla.Testa.EnableStopProgrammed )
   END_RUNG
   // the same network as SCL:
   #COut.Spalla.Testa.MoveToPos := #Ctrl.Spalle.Testa.MoveToPos;
   #COut.Spalla.Testa.Pos := #Ctrl.Spalle.Testa.Pos;
   #COut.Spalla.Testa.Speed := 30.0;
   #COut.Spalla.Testa.Control_ON := NOT (NOT #AreaInterface.Cycle AND NOT #Sts.SemiAut.ON);
   #COut.Spalla.Testa.EnableStopDoorOpeningReq := #MachineInterface.MotionsStandStill;
   #COut.Spalla.Testa.EnableStopInPhase := #MachineInterface.AckStopInPhase;
   #COut.Spalla.Testa.EnableStopProgrammed := #MachineInterface.AckStopProgrammed;
END_REGION

REGION Network 24: Spalla Coda - COut Manager
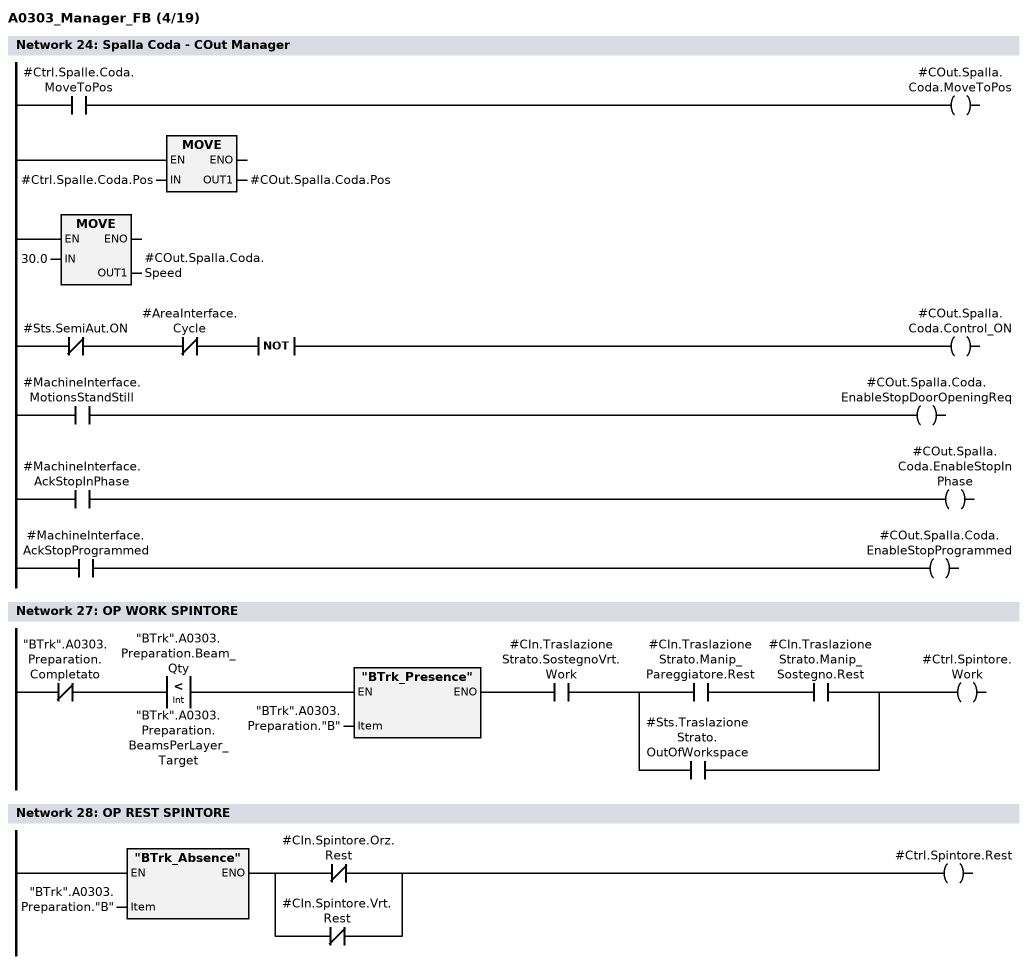
   RUNG wire#powerrail
      Contact( #Ctrl.Spalle.Coda.MoveToPos )
      Coil( #COut.Spalla.Coda.MoveToPos )
   END_RUNG
   RUNG wire#powerrail
      Move(in := #Ctrl.Spalle.Coda.Pos, out1 => #COut.Spalla.Coda.Pos)
   END_RUNG
   RUNG wire#powerrail
      Move(in := 30.0, out1 => #COut.Spalla.Coda.Speed)
   END_RUNG
   RUNG wire#powerrail
      I_Contact( #Sts.SemiAut.ON )
      I_Contact( #AreaInterface.Cycle )
      Not()
      Coil( #COut.Spalla.Coda.Control_ON )
   END_RUNG
   RUNG wire#powerrail
      Contact( #MachineInterface.MotionsStandStill )
      Coil( #COut.Spalla.Coda.EnableStopDoorOpeningReq )
   END_RUNG
   RUNG wire#powerrail
      Contact( #MachineInterface.AckStopInPhase )
      Coil( #COut.Spalla.Coda.EnableStopInPhase )
   END_RUNG
   RUNG wire#powerrail
      Contact( #MachineInterface.AckStopProgrammed )
      Coil( #COut.Spalla.Coda.EnableStopProgrammed )
   END_RUNG
   // the same network as SCL:
   #COut.Spalla.Coda.MoveToPos := #Ctrl.Spalle.Coda.MoveToPos;
   #COut.Spalla.Coda.Pos := #Ctrl.Spalle.Coda.Pos;
   #COut.Spalla.Coda.Speed := 30.0;
   #COut.Spalla.Coda.Control_ON := NOT (NOT #Sts.SemiAut.ON AND NOT #AreaInterface.Cycle);
   #COut.Spalla.Coda.EnableStopDoorOpeningReq := #MachineInterface.MotionsStandStill;
   #COut.Spalla.Coda.EnableStopInPhase := #MachineInterface.AckStopInPhase;
   #COut.Spalla.Coda.EnableStopProgrammed := #MachineInterface.AckStopProgrammed;
END_REGION

REGION Network 26: <<< SPINTORE STRATO >>>
END_REGION

REGION Network 27: OP WORK SPINTORE
   RUNG wire#powerrail
      I_Contact( "BTrk".A0303.Preparation.Completato )
      { S7_Templates := "SrcType := Int" } LT_Contact(in1 := "BTrk".A0303.Preparation.Beam_Qty, in2 := "BTrk".A0303.Preparation.BeamsPerLayer_Target)
      "BTrk_Presence"(Item := "BTrk".A0303.Preparation."B")
      Contact( #CIn.TraslazioneStrato.SostegnoVrt.Work )
      wire#w1
      Contact( #CIn.TraslazioneStrato.Manip_Pareggiatore.Rest )
      Contact( #CIn.TraslazioneStrato.Manip_Sostegno.Rest )
      wire#w2
      Coil( #Ctrl.Spintore.Work )
   END_RUNG
   RUNG wire#w1
      Contact( #Sts.TraslazioneStrato.OutOfWorkspace )
   END_RUNG wire#w2
   // the same network as SCL:
   "BTrk_Presence"(EN := NOT "BTrk".A0303.Preparation.Completato AND ("BTrk".A0303.Preparation.Beam_Qty < "BTrk".A0303.Preparation.BeamsPerLayer_Target),
                   Item := "BTrk".A0303.Preparation."B",
                   ENO => #_w1);
   #Ctrl.Spintore.Work := #_w1 AND #CIn.TraslazioneStrato.SostegnoVrt.Work AND ((#CIn.TraslazioneStrato.Manip_Pareggiatore.Rest AND #CIn.TraslazioneStrato.Manip_Sostegno.Rest) OR #Sts.TraslazioneStrato.OutOfWorkspace);
END_REGION

REGION Network 28: OP REST SPINTORE
   RUNG wire#powerrail
      "BTrk_Absence"(Item := "BTrk".A0303.Preparation."B")
      wire#w1
      I_Contact( #CIn.Spintore.Orz.Rest )
      wire#w2
      Coil( #Ctrl.Spintore.Rest )
   END_RUNG
   RUNG wire#w1
      I_Contact( #CIn.Spintore.Vrt.Rest )
   END_RUNG wire#w2
   // the same network as SCL:
   "BTrk_Absence"(Item := "BTrk".A0303.Preparation."B", ENO => #_w1);
   #Ctrl.Spintore.Rest := #_w1 AND (NOT #CIn.Spintore.Orz.Rest OR NOT #CIn.Spintore.Vrt.Rest);
END_REGION

REGION Network 29: Spintore - COut Manager
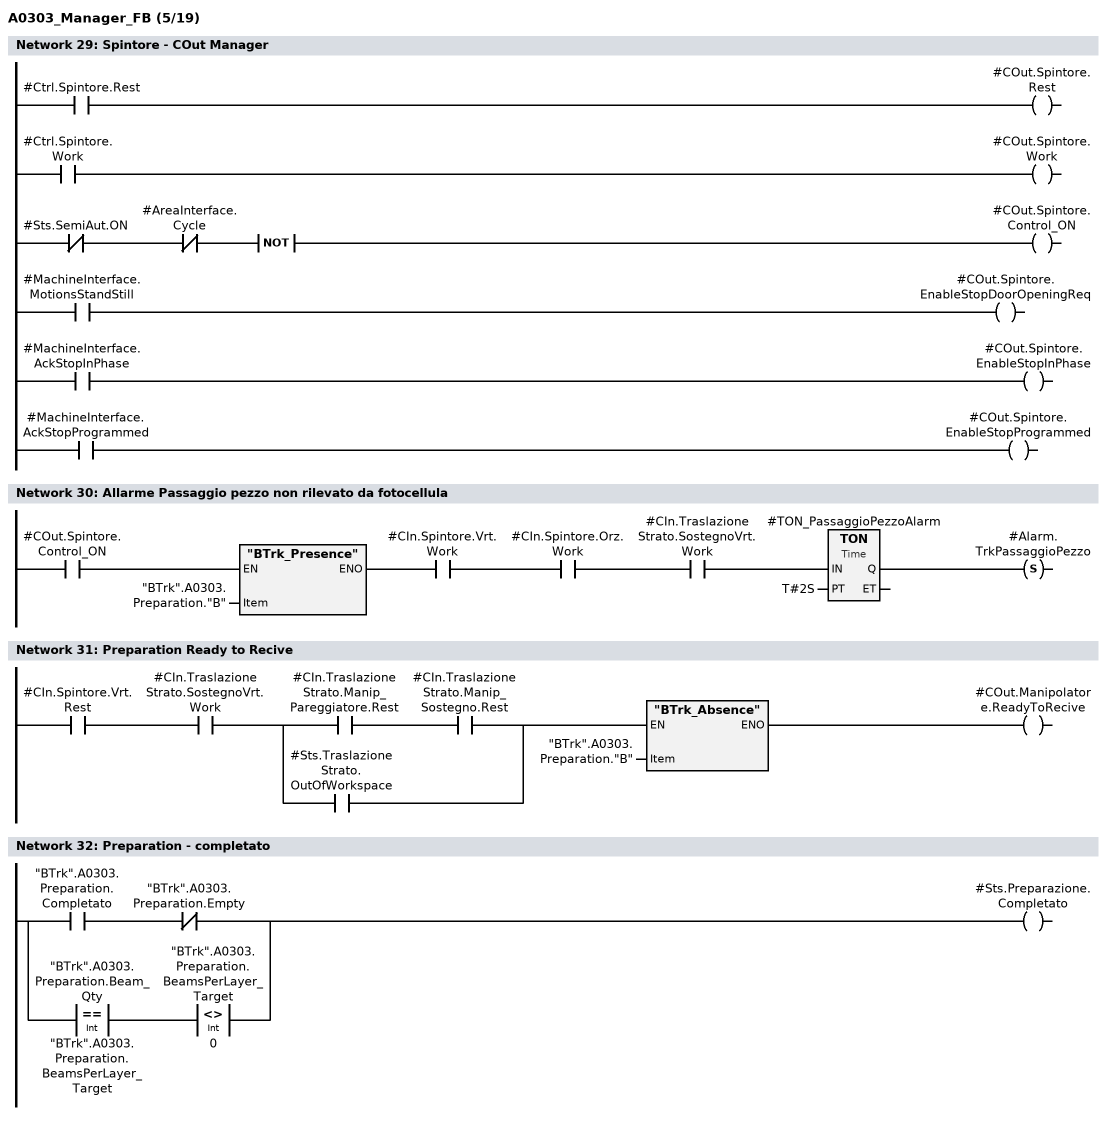
   RUNG wire#powerrail
      Contact( #Ctrl.Spintore.Rest )
      Coil( #COut.Spintore.Rest )
   END_RUNG
   RUNG wire#powerrail
      Contact( #Ctrl.Spintore.Work )
      Coil( #COut.Spintore.Work )
   END_RUNG
   RUNG wire#powerrail
      I_Contact( #Sts.SemiAut.ON )
      I_Contact( #AreaInterface.Cycle )
      Not()
      Coil( #COut.Spintore.Control_ON )
   END_RUNG
   RUNG wire#powerrail
      Contact( #MachineInterface.MotionsStandStill )
      Coil( #COut.Spintore.EnableStopDoorOpeningReq )
   END_RUNG
   RUNG wire#powerrail
      Contact( #MachineInterface.AckStopInPhase )
      Coil( #COut.Spintore.EnableStopInPhase )
   END_RUNG
   RUNG wire#powerrail
      Contact( #MachineInterface.AckStopProgrammed )
      Coil( #COut.Spintore.EnableStopProgrammed )
   END_RUNG
   // the same network as SCL:
   #COut.Spintore.Rest := #Ctrl.Spintore.Rest;
   #COut.Spintore.Work := #Ctrl.Spintore.Work;
   #COut.Spintore.Control_ON := NOT (NOT #Sts.SemiAut.ON AND NOT #AreaInterface.Cycle);
   #COut.Spintore.EnableStopDoorOpeningReq := #MachineInterface.MotionsStandStill;
   #COut.Spintore.EnableStopInPhase := #MachineInterface.AckStopInPhase;
   #COut.Spintore.EnableStopProgrammed := #MachineInterface.AckStopProgrammed;
END_REGION

REGION Network 30: Allarme Passaggio pezzo non rilevato da fotocellula
   RUNG wire#powerrail
      Contact( #COut.Spintore.Control_ON )
      "BTrk_Presence"(Item := "BTrk".A0303.Preparation."B")
      Contact( #CIn.Spintore.Vrt.Work )
      Contact( #CIn.Spintore.Orz.Work )
      Contact( #CIn.TraslazioneStrato.SostegnoVrt.Work )
      { S7_Templates := "time_type := Time" } #TON_PassaggioPezzoAlarm.TON(pt := T#2S, et =>)
      S_Coil( #Alarm.TrkPassaggioPezzo )
   END_RUNG
   // the same network as SCL:
   "BTrk_Presence"(EN := #COut.Spintore.Control_ON, Item := "BTrk".A0303.Preparation."B", ENO => #_w1);
   #TON_PassaggioPezzoAlarm.TON(IN := #_w1 AND #CIn.Spintore.Vrt.Work AND #CIn.Spintore.Orz.Work AND #CIn.TraslazioneStrato.SostegnoVrt.Work,
                           PT := T#2S);
   IF #TON_PassaggioPezzoAlarm.Q THEN #Alarm.TrkPassaggioPezzo := TRUE; END_IF;
END_REGION

REGION Network 31: Preparation Ready to Recive
   RUNG wire#powerrail
      Contact( #CIn.Spintore.Vrt.Rest )
      Contact( #CIn.TraslazioneStrato.SostegnoVrt.Work )
      wire#w1
      Contact( #CIn.TraslazioneStrato.Manip_Pareggiatore.Rest )
      Contact( #CIn.TraslazioneStrato.Manip_Sostegno.Rest )
      wire#w2
      "BTrk_Absence"(Item := "BTrk".A0303.Preparation."B")
      Coil( #COut.Manipolatore.ReadyToRecive )
   END_RUNG
   RUNG wire#w1
      Contact( #Sts.TraslazioneStrato.OutOfWorkspace )
   END_RUNG wire#w2
   // the same network as SCL:
   "BTrk_Absence"(EN := #CIn.Spintore.Vrt.Rest AND #CIn.TraslazioneStrato.SostegnoVrt.Work AND ((#CIn.TraslazioneStrato.Manip_Pareggiatore.Rest AND #CIn.TraslazioneStrato.Manip_Sostegno.Rest) OR #Sts.TraslazioneStrato.OutOfWorkspace),
                  Item := "BTrk".A0303.Preparation."B",
                  ENO => #_w1);
   #COut.Manipolatore.ReadyToRecive := #_w1;
END_REGION

REGION Network 32: Preparation - completato
   RUNG wire#powerrail
      Contact( "BTrk".A0303.Preparation.Completato )
      I_Contact( "BTrk".A0303.Preparation.Empty )
      wire#w1
      Coil( #Sts.Preparazione.Completato )
   END_RUNG
   RUNG wire#powerrail
      { S7_Templates := "SrcType := Int" } EQ_Contact(in1 := "BTrk".A0303.Preparation.Beam_Qty, in2 := "BTrk".A0303.Preparation.BeamsPerLayer_Target)
      { S7_Templates := "SrcType := Int" } NE_Contact(in1 := "BTrk".A0303.Preparation.BeamsPerLayer_Target, in2 := 0)
   END_RUNG wire#w1
   // the same network as SCL:
   #Sts.Preparazione.Completato := ("BTrk".A0303.Preparation.Completato AND NOT "BTrk".A0303.Preparation.Empty) OR (("BTrk".A0303.Preparation.Beam_Qty = "BTrk".A0303.Preparation.BeamsPerLayer_Target) AND ("BTrk".A0303.Preparation.BeamsPerLayer_Target <> 0));
END_REGION

REGION Network 33: <<<<<<<<<<<<<<<<<<<<<<<<<<<<<<<<<<< TRASFERIMENTO STRATO >>>>>>>>>>>>>>>>>>>>>>>>>>>>>>>>>>>>>>
END_REGION

REGION Network 34: Ax Trasporto in posizione
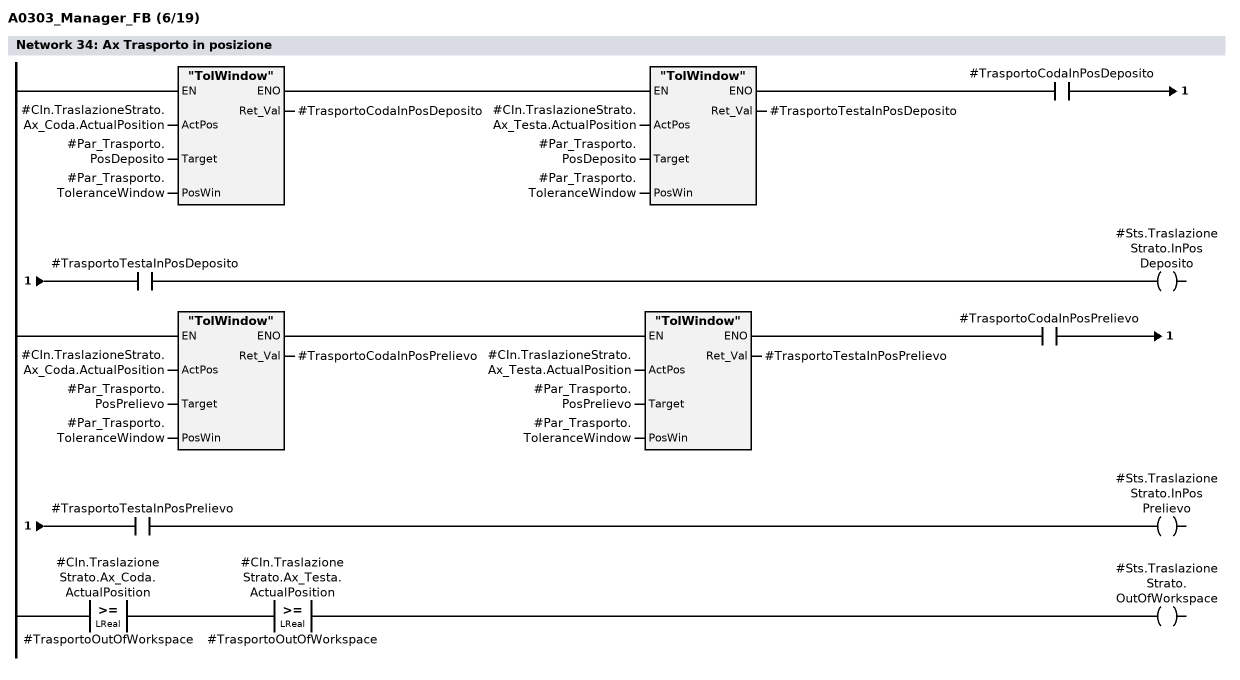
   RUNG wire#powerrail
      "TolWindow"(ActPos := #CIn.TraslazioneStrato.Ax_Coda.ActualPosition, Target := #Par_Trasporto.PosDeposito, PosWin := #Par_Trasporto.ToleranceWindow, Ret_Val => #TrasportoCodaInPosDeposito)
      "TolWindow"(ActPos := #CIn.TraslazioneStrato.Ax_Testa.ActualPosition, Target := #Par_Trasporto.PosDeposito, PosWin := #Par_Trasporto.ToleranceWindow, Ret_Val => #TrasportoTestaInPosDeposito)
      Contact( #TrasportoCodaInPosDeposito )
      Contact( #TrasportoTestaInPosDeposito )
      Coil( #Sts.TraslazioneStrato.InPosDeposito )
   END_RUNG
   RUNG wire#powerrail
      "TolWindow"(ActPos := #CIn.TraslazioneStrato.Ax_Coda.ActualPosition, Target := #Par_Trasporto.PosPrelievo, PosWin := #Par_Trasporto.ToleranceWindow, Ret_Val => #TrasportoCodaInPosPrelievo)
      "TolWindow"(ActPos := #CIn.TraslazioneStrato.Ax_Testa.ActualPosition, Target := #Par_Trasporto.PosPrelievo, PosWin := #Par_Trasporto.ToleranceWindow, Ret_Val => #TrasportoTestaInPosPrelievo)
      Contact( #TrasportoCodaInPosPrelievo )
      Contact( #TrasportoTestaInPosPrelievo )
      Coil( #Sts.TraslazioneStrato.InPosPrelievo )
   END_RUNG
   RUNG wire#powerrail
      { S7_Templates := "SrcType := LReal" } GE_Contact(in1 := #CIn.TraslazioneStrato.Ax_Coda.ActualPosition, in2 := #TrasportoOutOfWorkspace)
      { S7_Templates := "SrcType := LReal" } GE_Contact(in1 := #CIn.TraslazioneStrato.Ax_Testa.ActualPosition, in2 := #TrasportoOutOfWorkspace)
      Coil( #Sts.TraslazioneStrato.OutOfWorkspace )
   END_RUNG
   // the same network as SCL:
   #TrasportoCodaInPosDeposito := "TolWindow"(ActPos := #CIn.TraslazioneStrato.Ax_Coda.ActualPosition,
                           Target := #Par_Trasporto.PosDeposito,
                           PosWin := #Par_Trasporto.ToleranceWindow,
                           ENO => #_w1);
   #TrasportoTestaInPosDeposito := "TolWindow"(EN := #_w1,
                           ActPos := #CIn.TraslazioneStrato.Ax_Testa.ActualPosition,
                           Target := #Par_Trasporto.PosDeposito,
                           PosWin := #Par_Trasporto.ToleranceWindow,
                           ENO => #_w2);
   #Sts.TraslazioneStrato.InPosDeposito := #_w2 AND #TrasportoCodaInPosDeposito AND #TrasportoTestaInPosDeposito;
   #TrasportoCodaInPosPrelievo := "TolWindow"(ActPos := #CIn.TraslazioneStrato.Ax_Coda.ActualPosition,
                           Target := #Par_Trasporto.PosPrelievo,
                           PosWin := #Par_Trasporto.ToleranceWindow,
                           ENO => #_w3);
   #TrasportoTestaInPosPrelievo := "TolWindow"(EN := #_w3,
                           ActPos := #CIn.TraslazioneStrato.Ax_Testa.ActualPosition,
                           Target := #Par_Trasporto.PosPrelievo,
                           PosWin := #Par_Trasporto.ToleranceWindow,
                           ENO => #_w4);
   #Sts.TraslazioneStrato.InPosPrelievo := #_w4 AND #TrasportoCodaInPosPrelievo AND #TrasportoTestaInPosPrelievo;
   #Sts.TraslazioneStrato.OutOfWorkspace := (#CIn.TraslazioneStrato.Ax_Coda.ActualPosition >= #TrasportoOutOfWorkspace) AND (#CIn.TraslazioneStrato.Ax_Testa.ActualPosition >= #TrasportoOutOfWorkspace);
END_REGION

REGION Network 35: Fasi trasporto
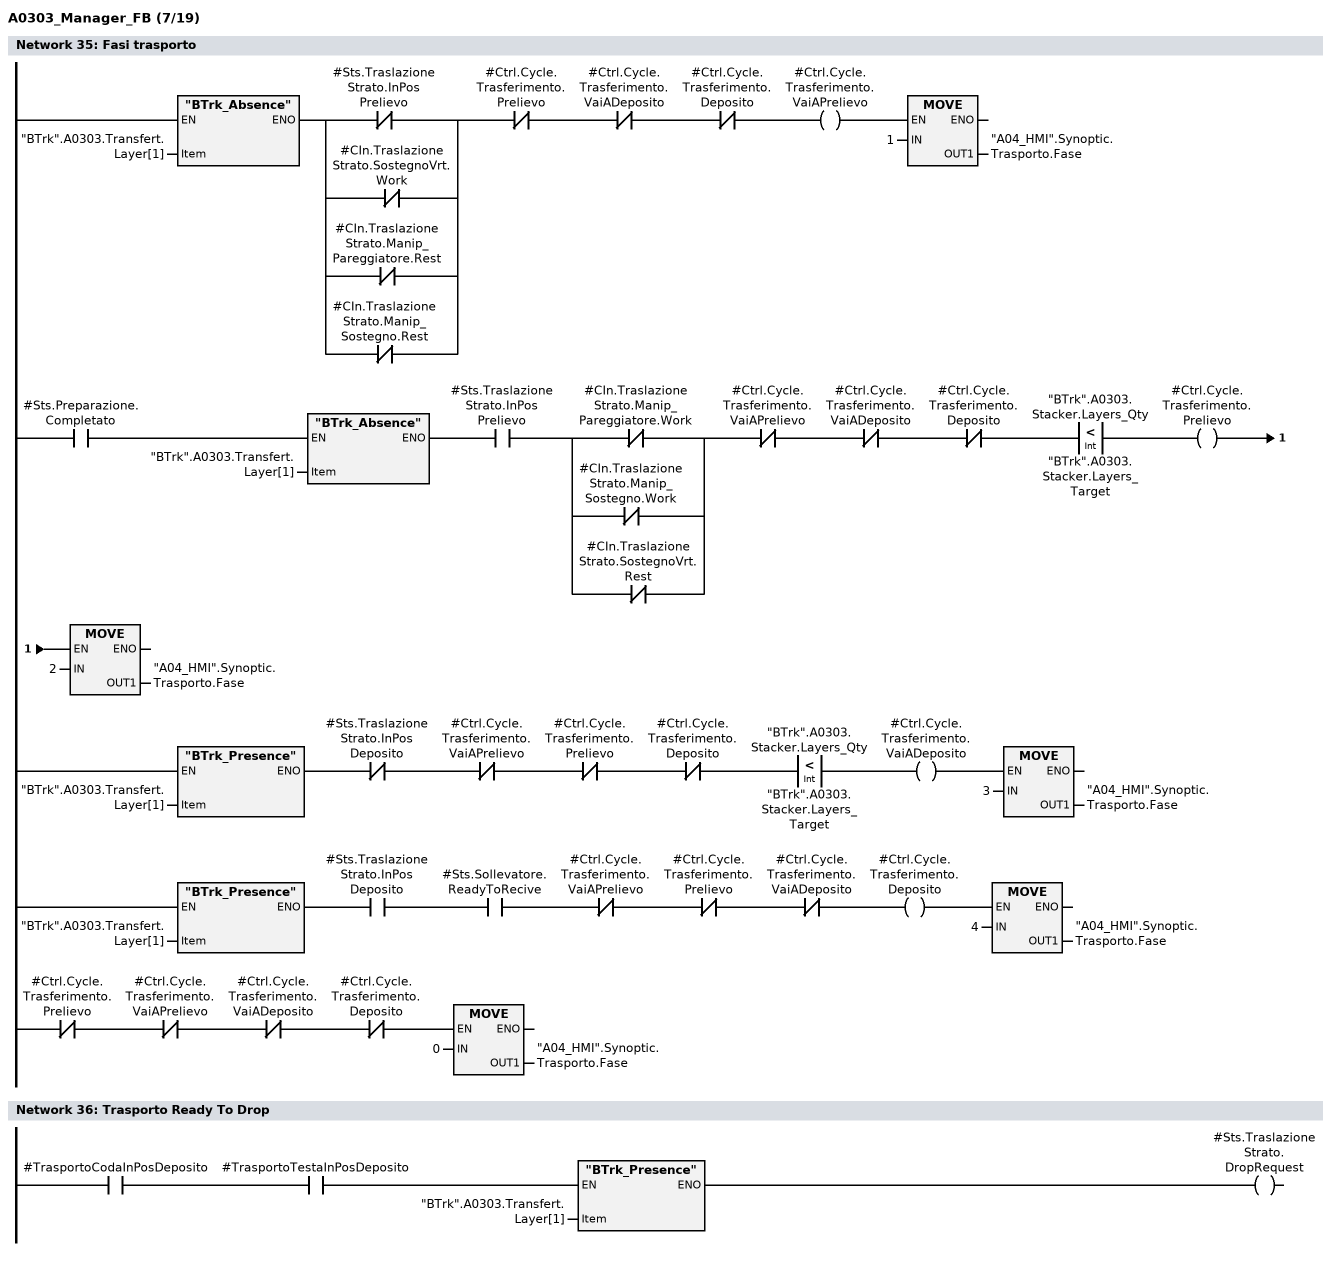
   RUNG wire#powerrail
      "BTrk_Absence"(Item := "BTrk".A0303.Transfert.Layer[1])
      wire#w1
      I_Contact( #Sts.TraslazioneStrato.InPosPrelievo )
      wire#w2
      I_Contact( #Ctrl.Cycle.Trasferimento.Prelievo )
      I_Contact( #Ctrl.Cycle.Trasferimento.VaiADeposito )
      I_Contact( #Ctrl.Cycle.Trasferimento.Deposito )
      Coil( #Ctrl.Cycle.Trasferimento.VaiAPrelievo )
      Move(in := 1, out1 => "A04_HMI".Synoptic.Trasporto.Fase)
   END_RUNG
   RUNG wire#w1
      I_Contact( #CIn.TraslazioneStrato.SostegnoVrt.Work )
   END_RUNG wire#w2
   RUNG wire#w1
      I_Contact( #CIn.TraslazioneStrato.Manip_Pareggiatore.Rest )
   END_RUNG wire#w2
   RUNG wire#w1
      I_Contact( #CIn.TraslazioneStrato.Manip_Sostegno.Rest )
   END_RUNG wire#w2
   RUNG wire#powerrail
      Contact( #Sts.Preparazione.Completato )
      "BTrk_Absence"(Item := "BTrk".A0303.Transfert.Layer[1])
      Contact( #Sts.TraslazioneStrato.InPosPrelievo )
      wire#w3
      I_Contact( #CIn.TraslazioneStrato.Manip_Pareggiatore.Work )
      wire#w4
      I_Contact( #Ctrl.Cycle.Trasferimento.VaiAPrelievo )
      I_Contact( #Ctrl.Cycle.Trasferimento.VaiADeposito )
      I_Contact( #Ctrl.Cycle.Trasferimento.Deposito )
      { S7_Templates := "SrcType := Int" } LT_Contact(in1 := "BTrk".A0303.Stacker.Layers_Qty, in2 := "BTrk".A0303.Stacker.Layers_Target)
      Coil( #Ctrl.Cycle.Trasferimento.Prelievo )
      Move(in := 2, out1 => "A04_HMI".Synoptic.Trasporto.Fase)
   END_RUNG
   RUNG wire#w3
      I_Contact( #CIn.TraslazioneStrato.Manip_Sostegno.Work )
   END_RUNG wire#w4
   RUNG wire#w3
      I_Contact( #CIn.TraslazioneStrato.SostegnoVrt.Rest )
   END_RUNG wire#w4
   RUNG wire#powerrail
      "BTrk_Presence"(Item := "BTrk".A0303.Transfert.Layer[1])
      I_Contact( #Sts.TraslazioneStrato.InPosDeposito )
      I_Contact( #Ctrl.Cycle.Trasferimento.VaiAPrelievo )
      I_Contact( #Ctrl.Cycle.Trasferimento.Prelievo )
      I_Contact( #Ctrl.Cycle.Trasferimento.Deposito )
      { S7_Templates := "SrcType := Int" } LT_Contact(in1 := "BTrk".A0303.Stacker.Layers_Qty, in2 := "BTrk".A0303.Stacker.Layers_Target)
      Coil( #Ctrl.Cycle.Trasferimento.VaiADeposito )
      Move(in := 3, out1 => "A04_HMI".Synoptic.Trasporto.Fase)
   END_RUNG
   RUNG wire#powerrail
      "BTrk_Presence"(Item := "BTrk".A0303.Transfert.Layer[1])
      Contact( #Sts.TraslazioneStrato.InPosDeposito )
      Contact( #Sts.Sollevatore.ReadyToRecive )
      I_Contact( #Ctrl.Cycle.Trasferimento.VaiAPrelievo )
      I_Contact( #Ctrl.Cycle.Trasferimento.Prelievo )
      I_Contact( #Ctrl.Cycle.Trasferimento.VaiADeposito )
      Coil( #Ctrl.Cycle.Trasferimento.Deposito )
      Move(in := 4, out1 => "A04_HMI".Synoptic.Trasporto.Fase)
   END_RUNG
   RUNG wire#powerrail
      I_Contact( #Ctrl.Cycle.Trasferimento.Prelievo )
      I_Contact( #Ctrl.Cycle.Trasferimento.VaiAPrelievo )
      I_Contact( #Ctrl.Cycle.Trasferimento.VaiADeposito )
      I_Contact( #Ctrl.Cycle.Trasferimento.Deposito )
      Move(in := 0, out1 => "A04_HMI".Synoptic.Trasporto.Fase)
   END_RUNG
   // the same network as SCL:
   "BTrk_Absence"(Item := "BTrk".A0303.Transfert.Layer[1], ENO => #_w1);
   #Ctrl.Cycle.Trasferimento.VaiAPrelievo := #_w1 AND (NOT #Sts.TraslazioneStrato.InPosPrelievo OR NOT #CIn.TraslazioneStrato.SostegnoVrt.Work OR NOT #CIn.TraslazioneStrato.Manip_Pareggiatore.Rest OR NOT #CIn.TraslazioneStrato.Manip_Sostegno.Rest) AND NOT #Ctrl.Cycle.Trasferimento.Prelievo AND NOT #Ctrl.Cycle.Trasferimento.VaiADeposito AND NOT #Ctrl.Cycle.Trasferimento.Deposito;
   IF #Ctrl.Cycle.Trasferimento.VaiAPrelievo THEN "A04_HMI".Synoptic.Trasporto.Fase := 1; END_IF;
   "BTrk_Absence"(EN := #Sts.Preparazione.Completato, Item := "BTrk".A0303.Transfert.Layer[1], ENO => #_w2);
   #Ctrl.Cycle.Trasferimento.Prelievo := #_w2 AND #Sts.TraslazioneStrato.InPosPrelievo AND (NOT #CIn.TraslazioneStrato.Manip_Pareggiatore.Work OR NOT #CIn.TraslazioneStrato.Manip_Sostegno.Work OR NOT #CIn.TraslazioneStrato.SostegnoVrt.Rest) AND NOT #Ctrl.Cycle.Trasferimento.VaiAPrelievo AND NOT #Ctrl.Cycle.Trasferimento.VaiADeposito AND NOT #Ctrl.Cycle.Trasferimento.Deposito AND ("BTrk".A0303.Stacker.Layers_Qty < "BTrk".A0303.Stacker.Layers_Target);
   IF #Ctrl.Cycle.Trasferimento.Prelievo THEN "A04_HMI".Synoptic.Trasporto.Fase := 2; END_IF;
   "BTrk_Presence"(Item := "BTrk".A0303.Transfert.Layer[1], ENO => #_w3);
   #Ctrl.Cycle.Trasferimento.VaiADeposito := #_w3 AND NOT #Sts.TraslazioneStrato.InPosDeposito AND NOT #Ctrl.Cycle.Trasferimento.VaiAPrelievo AND NOT #Ctrl.Cycle.Trasferimento.Prelievo AND NOT #Ctrl.Cycle.Trasferimento.Deposito AND ("BTrk".A0303.Stacker.Layers_Qty < "BTrk".A0303.Stacker.Layers_Target);
   IF #Ctrl.Cycle.Trasferimento.VaiADeposito THEN "A04_HMI".Synoptic.Trasporto.Fase := 3; END_IF;
   "BTrk_Presence"(Item := "BTrk".A0303.Transfert.Layer[1], ENO => #_w4);
   #Ctrl.Cycle.Trasferimento.Deposito := #_w4 AND #Sts.TraslazioneStrato.InPosDeposito AND #Sts.Sollevatore.ReadyToRecive AND NOT #Ctrl.Cycle.Trasferimento.VaiAPrelievo AND NOT #Ctrl.Cycle.Trasferimento.Prelievo AND NOT #Ctrl.Cycle.Trasferimento.VaiADeposito;
   IF #Ctrl.Cycle.Trasferimento.Deposito THEN "A04_HMI".Synoptic.Trasporto.Fase := 4; END_IF;
   IF NOT #Ctrl.Cycle.Trasferimento.Prelievo AND NOT #Ctrl.Cycle.Trasferimento.VaiAPrelievo AND NOT #Ctrl.Cycle.Trasferimento.VaiADeposito AND NOT #Ctrl.Cycle.Trasferimento.Deposito THEN
       "A04_HMI".Synoptic.Trasporto.Fase := 0;
   END_IF;
END_REGION

REGION Network 36: Trasporto Ready To Drop
   RUNG wire#powerrail
      Contact( #TrasportoCodaInPosDeposito )
      Contact( #TrasportoTestaInPosDeposito )
      "BTrk_Presence"(Item := "BTrk".A0303.Transfert.Layer[1])
      Coil( #Sts.TraslazioneStrato.DropRequest )
   END_RUNG
   // the same network as SCL:
   "BTrk_Presence"(EN := #TrasportoCodaInPosDeposito AND #TrasportoTestaInPosDeposito,
                   Item := "BTrk".A0303.Transfert.Layer[1],
                   ENO => #_w1);
   #Sts.TraslazioneStrato.DropRequest := #_w1;
END_REGION

REGION Network 37: Trasporto - COut Manager
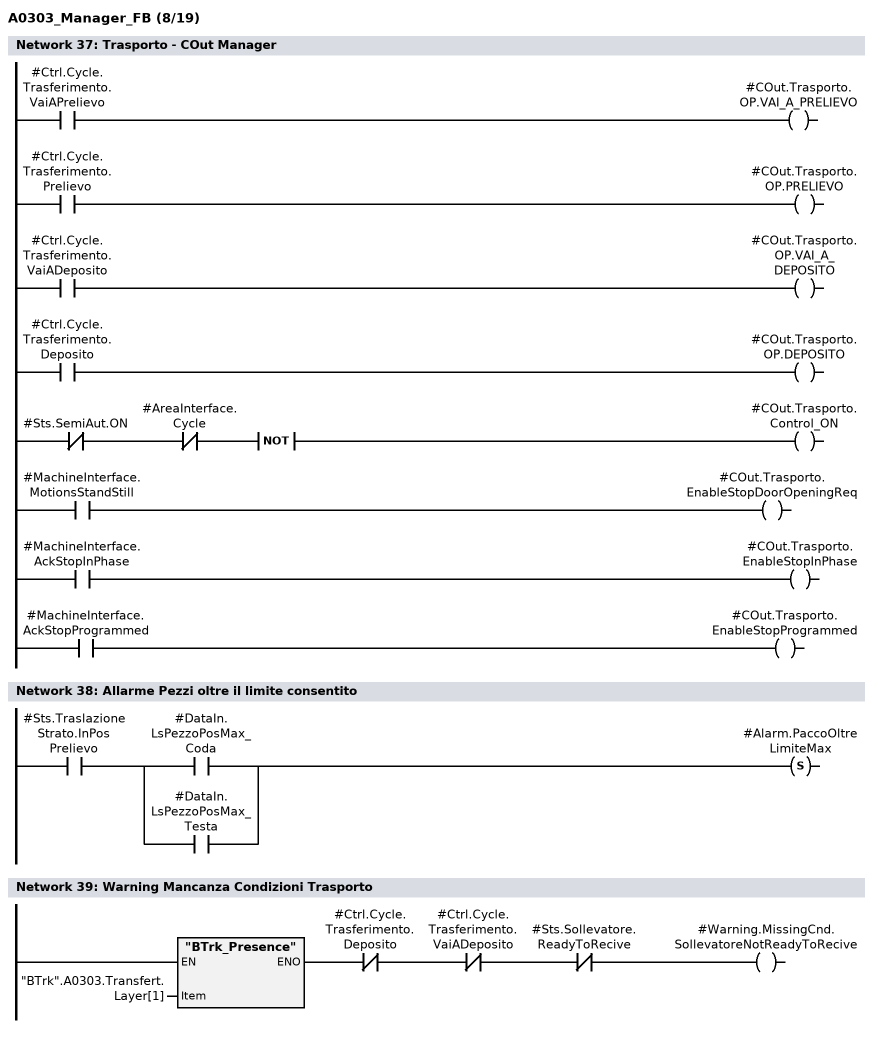
   RUNG wire#powerrail
      Contact( #Ctrl.Cycle.Trasferimento.VaiAPrelievo )
      Coil( #COut.Trasporto.OP.VAI_A_PRELIEVO )
   END_RUNG
   RUNG wire#powerrail
      Contact( #Ctrl.Cycle.Trasferimento.Prelievo )
      Coil( #COut.Trasporto.OP.PRELIEVO )
   END_RUNG
   RUNG wire#powerrail
      Contact( #Ctrl.Cycle.Trasferimento.VaiADeposito )
      Coil( #COut.Trasporto.OP.VAI_A_DEPOSITO )
   END_RUNG
   RUNG wire#powerrail
      Contact( #Ctrl.Cycle.Trasferimento.Deposito )
      Coil( #COut.Trasporto.OP.DEPOSITO )
   END_RUNG
   RUNG wire#powerrail
      I_Contact( #Sts.SemiAut.ON )
      I_Contact( #AreaInterface.Cycle )
      Not()
      Coil( #COut.Trasporto.Control_ON )
   END_RUNG
   RUNG wire#powerrail
      Contact( #MachineInterface.MotionsStandStill )
      Coil( #COut.Trasporto.EnableStopDoorOpeningReq )
   END_RUNG
   RUNG wire#powerrail
      Contact( #MachineInterface.AckStopInPhase )
      Coil( #COut.Trasporto.EnableStopInPhase )
   END_RUNG
   RUNG wire#powerrail
      Contact( #MachineInterface.AckStopProgrammed )
      Coil( #COut.Trasporto.EnableStopProgrammed )
   END_RUNG
   // the same network as SCL:
   #COut.Trasporto.OP.VAI_A_PRELIEVO := #Ctrl.Cycle.Trasferimento.VaiAPrelievo;
   #COut.Trasporto.OP.PRELIEVO := #Ctrl.Cycle.Trasferimento.Prelievo;
   #COut.Trasporto.OP.VAI_A_DEPOSITO := #Ctrl.Cycle.Trasferimento.VaiADeposito;
   #COut.Trasporto.OP.DEPOSITO := #Ctrl.Cycle.Trasferimento.Deposito;
   #COut.Trasporto.Control_ON := NOT (NOT #Sts.SemiAut.ON AND NOT #AreaInterface.Cycle);
   #COut.Trasporto.EnableStopDoorOpeningReq := #MachineInterface.MotionsStandStill;
   #COut.Trasporto.EnableStopInPhase := #MachineInterface.AckStopInPhase;
   #COut.Trasporto.EnableStopProgrammed := #MachineInterface.AckStopProgrammed;
END_REGION

REGION Network 38: Allarme Pezzi oltre il limite consentito
   RUNG wire#powerrail
      Contact( #Sts.TraslazioneStrato.InPosPrelievo )
      wire#w1
      Contact( #DataIn.LsPezzoPosMax_Coda )
      wire#w2
      S_Coil( #Alarm.PaccoOltreLimiteMax )
   END_RUNG
   RUNG wire#w1
      Contact( #DataIn.LsPezzoPosMax_Testa )
   END_RUNG wire#w2
   // the same network as SCL:
   IF #Sts.TraslazioneStrato.InPosPrelievo AND (#DataIn.LsPezzoPosMax_Coda OR #DataIn.LsPezzoPosMax_Testa) THEN
       #Alarm.PaccoOltreLimiteMax := TRUE;
   END_IF;
END_REGION

REGION Network 39: Warning Mancanza Condizioni Trasporto
   RUNG wire#powerrail
      "BTrk_Presence"(Item := "BTrk".A0303.Transfert.Layer[1])
      I_Contact( #Ctrl.Cycle.Trasferimento.Deposito )
      I_Contact( #Ctrl.Cycle.Trasferimento.VaiADeposito )
      I_Contact( #Sts.Sollevatore.ReadyToRecive )
      Coil( #Warning.MissingCnd.SollevatoreNotReadyToRecive )
   END_RUNG
   // the same network as SCL:
   "BTrk_Presence"(Item := "BTrk".A0303.Transfert.Layer[1], ENO => #_w1);
   #Warning.MissingCnd.SollevatoreNotReadyToRecive := #_w1 AND NOT #Ctrl.Cycle.Trasferimento.Deposito AND NOT #Ctrl.Cycle.Trasferimento.VaiADeposito AND NOT #Sts.Sollevatore.ReadyToRecive;
END_REGION

REGION Network 40: <<<<<<<<<<<<<<<<<<<<<<<<<<<<<<<<<<<<<<<<< IMPILAMENTO >>>>>>>>>>>>>>>>>>>>>>>>>>>>>>>>>>>>>>>>>>>
END_REGION

REGION Network 41: <<< SOLLEVATORE >>>
END_REGION

REGION Network 42: Calcolo Target di posizionamento
   // Finche non c'è la richiesta di scaricare il pezzo il sollevatore si porta un po piu basso ad una quota di pre prelievo, quando poi c'è la richiesta di scaricare il pezzo si alza di un offset
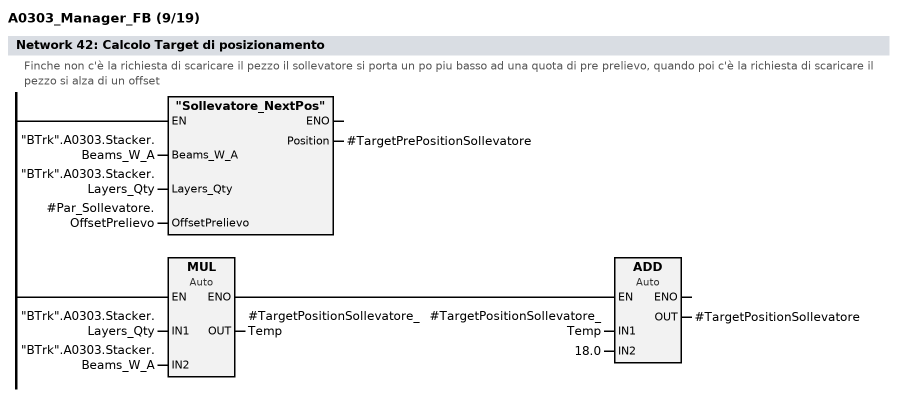
   RUNG wire#powerrail
      "Sollevatore_NextPos"(Beams_W_A := "BTrk".A0303.Stacker.Beams_W_A, Layers_Qty := "BTrk".A0303.Stacker.Layers_Qty, OffsetPrelievo := #Par_Sollevatore.OffsetPrelievo, Position => #TargetPrePositionSollevatore)
   END_RUNG
   RUNG wire#powerrail
      Mul(in1 := "BTrk".A0303.Stacker.Layers_Qty, in2 := "BTrk".A0303.Stacker.Beams_W_A, out => #TargetPositionSollevatore_Temp)
      Add(in1 := #TargetPositionSollevatore_Temp, in2 := 18.0, out => #TargetPositionSollevatore)
   END_RUNG
   // the same network as SCL:
   "Sollevatore_NextPos"(Beams_W_A := "BTrk".A0303.Stacker.Beams_W_A,
                         Layers_Qty := "BTrk".A0303.Stacker.Layers_Qty,
                         OffsetPrelievo := #Par_Sollevatore.OffsetPrelievo,
                         Position => #TargetPrePositionSollevatore);
   #TargetPositionSollevatore_Temp := "BTrk".A0303.Stacker.Layers_Qty * "BTrk".A0303.Stacker.Beams_W_A;
   #TargetPositionSollevatore := #TargetPositionSollevatore_Temp + 18.0;
END_REGION

REGION Network 43: Ax position window
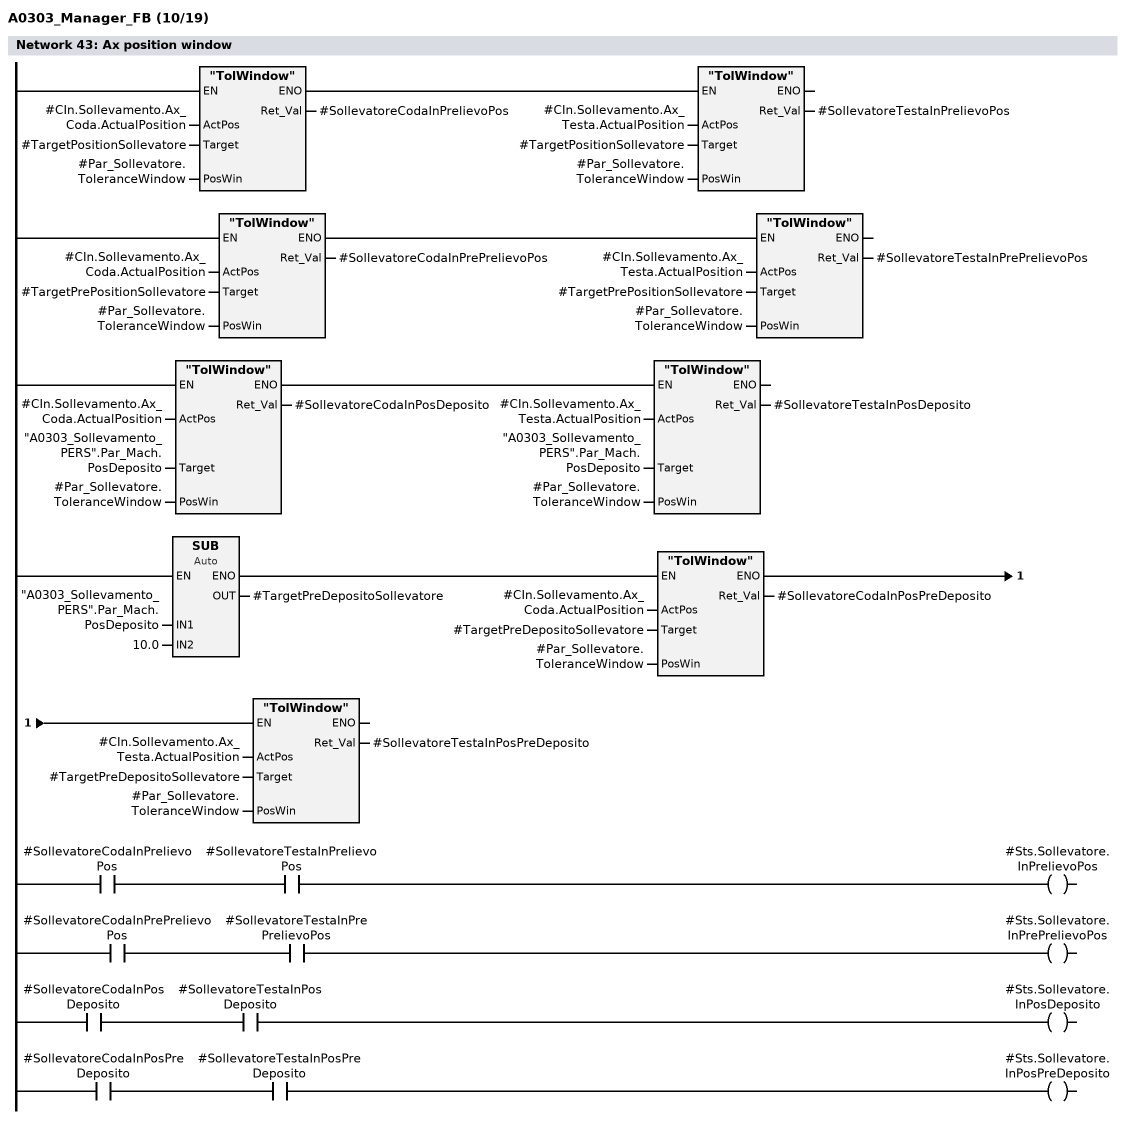
   RUNG wire#powerrail
      "TolWindow"(ActPos := #CIn.Sollevamento.Ax_Coda.ActualPosition, Target := #TargetPositionSollevatore, PosWin := #Par_Sollevatore.ToleranceWindow, Ret_Val => #SollevatoreCodaInPrelievoPos)
      "TolWindow"(ActPos := #CIn.Sollevamento.Ax_Testa.ActualPosition, Target := #TargetPositionSollevatore, PosWin := #Par_Sollevatore.ToleranceWindow, Ret_Val => #SollevatoreTestaInPrelievoPos)
   END_RUNG
   RUNG wire#powerrail
      "TolWindow"(ActPos := #CIn.Sollevamento.Ax_Coda.ActualPosition, Target := #TargetPrePositionSollevatore, PosWin := #Par_Sollevatore.ToleranceWindow, Ret_Val => #SollevatoreCodaInPrePrelievoPos)
      "TolWindow"(ActPos := #CIn.Sollevamento.Ax_Testa.ActualPosition, Target := #TargetPrePositionSollevatore, PosWin := #Par_Sollevatore.ToleranceWindow, Ret_Val => #SollevatoreTestaInPrePrelievoPos)
   END_RUNG
   RUNG wire#powerrail
      "TolWindow"(ActPos := #CIn.Sollevamento.Ax_Coda.ActualPosition, Target := "A0303_Sollevamento_PERS".Par_Mach.PosDeposito, PosWin := #Par_Sollevatore.ToleranceWindow, Ret_Val => #SollevatoreCodaInPosDeposito)
      "TolWindow"(ActPos := #CIn.Sollevamento.Ax_Testa.ActualPosition, Target := "A0303_Sollevamento_PERS".Par_Mach.PosDeposito, PosWin := #Par_Sollevatore.ToleranceWindow, Ret_Val => #SollevatoreTestaInPosDeposito)
   END_RUNG
   RUNG wire#powerrail
      Sub(in1 := "A0303_Sollevamento_PERS".Par_Mach.PosDeposito, in2 := 10.0, out => #TargetPreDepositoSollevatore)
      "TolWindow"(ActPos := #CIn.Sollevamento.Ax_Coda.ActualPosition, Target := #TargetPreDepositoSollevatore, PosWin := #Par_Sollevatore.ToleranceWindow, Ret_Val => #SollevatoreCodaInPosPreDeposito)
      "TolWindow"(ActPos := #CIn.Sollevamento.Ax_Testa.ActualPosition, Target := #TargetPreDepositoSollevatore, PosWin := #Par_Sollevatore.ToleranceWindow, Ret_Val => #SollevatoreTestaInPosPreDeposito)
   END_RUNG
   RUNG wire#powerrail
      Contact( #SollevatoreCodaInPrelievoPos )
      Contact( #SollevatoreTestaInPrelievoPos )
      Coil( #Sts.Sollevatore.InPrelievoPos )
   END_RUNG
   RUNG wire#powerrail
      Contact( #SollevatoreCodaInPrePrelievoPos )
      Contact( #SollevatoreTestaInPrePrelievoPos )
      Coil( #Sts.Sollevatore.InPrePrelievoPos )
   END_RUNG
   RUNG wire#powerrail
      Contact( #SollevatoreCodaInPosDeposito )
      Contact( #SollevatoreTestaInPosDeposito )
      Coil( #Sts.Sollevatore.InPosDeposito )
   END_RUNG
   RUNG wire#powerrail
      Contact( #SollevatoreCodaInPosPreDeposito )
      Contact( #SollevatoreTestaInPosPreDeposito )
      Coil( #Sts.Sollevatore.InPosPreDeposito )
   END_RUNG
   // the same network as SCL:
   #SollevatoreCodaInPrelievoPos := "TolWindow"(ActPos := #CIn.Sollevamento.Ax_Coda.ActualPosition,
                           Target := #TargetPositionSollevatore,
                           PosWin := #Par_Sollevatore.ToleranceWindow,
                           ENO => #_w1);
   IF #_w1 THEN
       #SollevatoreTestaInPrelievoPos := "TolWindow"(ActPos := #CIn.Sollevamento.Ax_Testa.ActualPosition,
                               Target := #TargetPositionSollevatore,
                               PosWin := #Par_Sollevatore.ToleranceWindow);
   END_IF;
   #SollevatoreCodaInPrePrelievoPos := "TolWindow"(ActPos := #CIn.Sollevamento.Ax_Coda.ActualPosition,
                           Target := #TargetPrePositionSollevatore,
                           PosWin := #Par_Sollevatore.ToleranceWindow,
                           ENO => #_w2);
   IF #_w2 THEN
       #SollevatoreTestaInPrePrelievoPos := "TolWindow"(ActPos := #CIn.Sollevamento.Ax_Testa.ActualPosition,
                               Target := #TargetPrePositionSollevatore,
                               PosWin := #Par_Sollevatore.ToleranceWindow);
   END_IF;
   #SollevatoreCodaInPosDeposito := "TolWindow"(ActPos := #CIn.Sollevamento.Ax_Coda.ActualPosition,
                           Target := "A0303_Sollevamento_PERS".Par_Mach.PosDeposito,
                           PosWin := #Par_Sollevatore.ToleranceWindow,
                           ENO => #_w3);
   IF #_w3 THEN
       #SollevatoreTestaInPosDeposito := "TolWindow"(ActPos := #CIn.Sollevamento.Ax_Testa.ActualPosition,
                               Target := "A0303_Sollevamento_PERS".Par_Mach.PosDeposito,
                               PosWin := #Par_Sollevatore.ToleranceWindow);
   END_IF;
   #TargetPreDepositoSollevatore := "A0303_Sollevamento_PERS".Par_Mach.PosDeposito - 10.0;
   #SollevatoreCodaInPosPreDeposito := "TolWindow"(ActPos := #CIn.Sollevamento.Ax_Coda.ActualPosition,
                           Target := #TargetPreDepositoSollevatore,
                           PosWin := #Par_Sollevatore.ToleranceWindow,
                           ENO => #_w4);
   IF #_w4 THEN
       #SollevatoreTestaInPosPreDeposito := "TolWindow"(ActPos := #CIn.Sollevamento.Ax_Testa.ActualPosition,
                               Target := #TargetPreDepositoSollevatore,
                               PosWin := #Par_Sollevatore.ToleranceWindow);
   END_IF;
   #Sts.Sollevatore.InPrelievoPos := #SollevatoreCodaInPrelievoPos AND #SollevatoreTestaInPrelievoPos;
   #Sts.Sollevatore.InPrePrelievoPos := #SollevatoreCodaInPrePrelievoPos AND #SollevatoreTestaInPrePrelievoPos;
   #Sts.Sollevatore.InPosDeposito := #SollevatoreCodaInPosDeposito AND #SollevatoreTestaInPosDeposito;
   #Sts.Sollevatore.InPosPreDeposito := #SollevatoreCodaInPosPreDeposito AND #SollevatoreTestaInPosPreDeposito;
END_REGION

REGION Network 44: Fasi Sollevatore
   // Fasi Sollevatore : Il sollevatore si deve portare in posizione di preprelievo e quando il traslatore è in posizione di deposito e pronto a depositare allora posso salire e  prelevare il pezzo
   // Quando raggiungo il numero max di layer passo alla fase di deposito
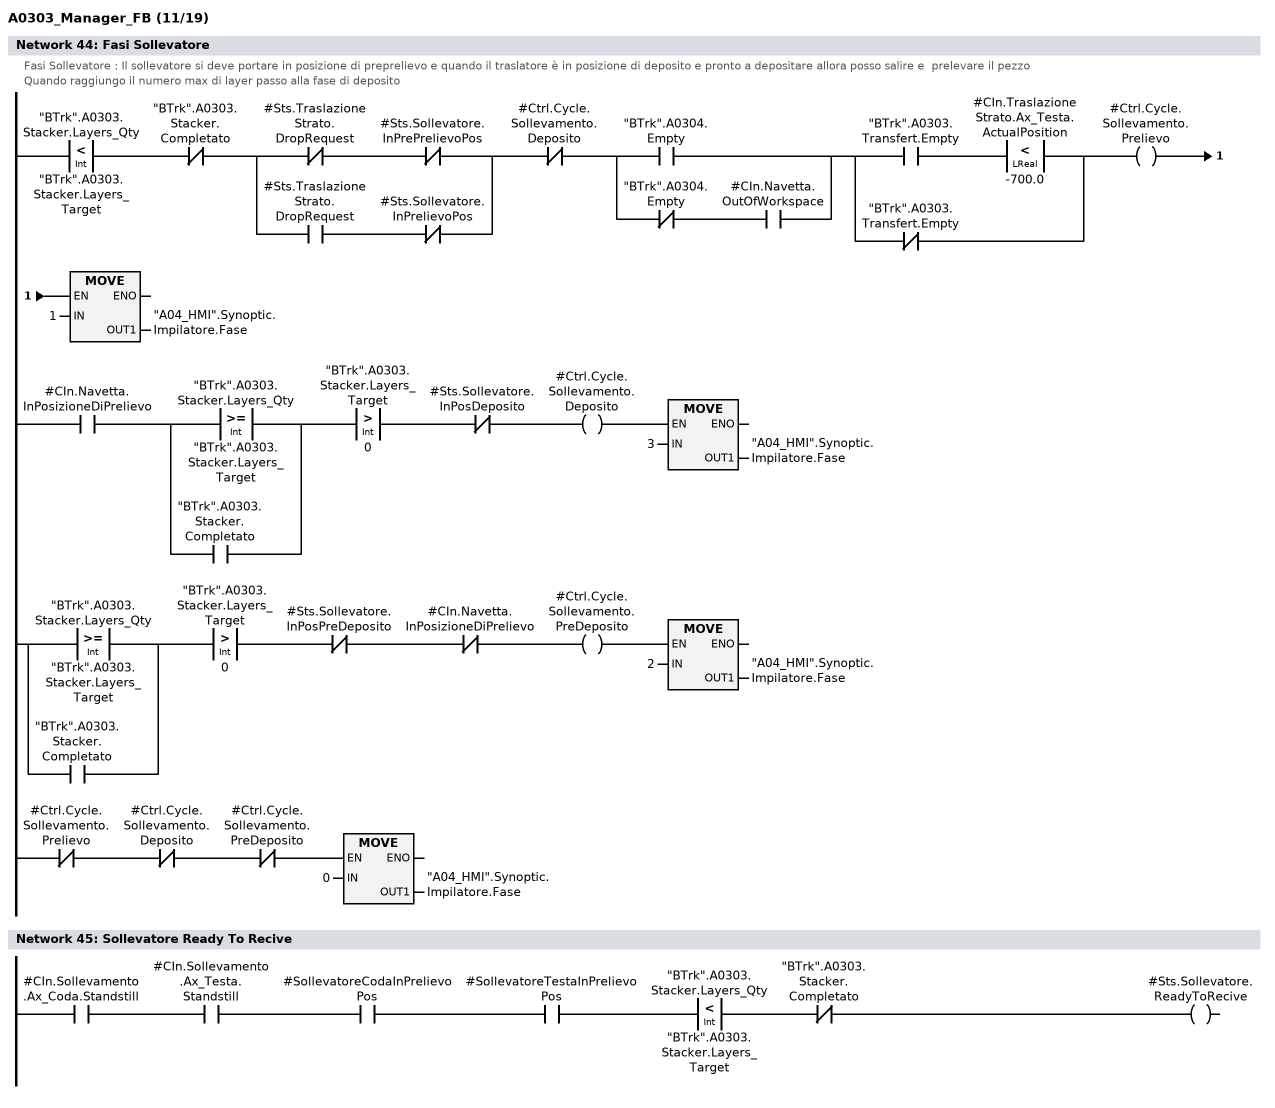
   RUNG wire#powerrail
      { S7_Templates := "SrcType := Int" } LT_Contact(in1 := "BTrk".A0303.Stacker.Layers_Qty, in2 := "BTrk".A0303.Stacker.Layers_Target)
      I_Contact( "BTrk".A0303.Stacker.Completato )
      wire#w1
      I_Contact( #Sts.TraslazioneStrato.DropRequest )
      I_Contact( #Sts.Sollevatore.InPrePrelievoPos )
      wire#w2
      I_Contact( #Ctrl.Cycle.Sollevamento.Deposito )
      wire#w3
      Contact( "BTrk".A0304.Empty )
      wire#w4
      Contact( "BTrk".A0303.Transfert.Empty )
      { S7_Templates := "SrcType := LReal" } LT_Contact(in1 := #CIn.TraslazioneStrato.Ax_Testa.ActualPosition, in2 := -700.0)
      wire#w5
      Coil( #Ctrl.Cycle.Sollevamento.Prelievo )
      Move(in := 1, out1 => "A04_HMI".Synoptic.Impilatore.Fase)
   END_RUNG
   RUNG wire#w1
      Contact( #Sts.TraslazioneStrato.DropRequest )
      I_Contact( #Sts.Sollevatore.InPrelievoPos )
   END_RUNG wire#w2
   RUNG wire#w3
      I_Contact( "BTrk".A0304.Empty )
      Contact( #CIn.Navetta.OutOfWorkspace )
   END_RUNG wire#w4
   RUNG wire#w4
      I_Contact( "BTrk".A0303.Transfert.Empty )
   END_RUNG wire#w5
   RUNG wire#powerrail
      Contact( #CIn.Navetta.InPosizioneDiPrelievo )
      wire#w6
      { S7_Templates := "SrcType := Int" } GE_Contact(in1 := "BTrk".A0303.Stacker.Layers_Qty, in2 := "BTrk".A0303.Stacker.Layers_Target)
      wire#w7
      { S7_Templates := "SrcType := Int" } GT_Contact(in1 := "BTrk".A0303.Stacker.Layers_Target, in2 := 0)
      I_Contact( #Sts.Sollevatore.InPosDeposito )
      Coil( #Ctrl.Cycle.Sollevamento.Deposito )
      Move(in := 3, out1 => "A04_HMI".Synoptic.Impilatore.Fase)
   END_RUNG
   RUNG wire#w6
      Contact( "BTrk".A0303.Stacker.Completato )
   END_RUNG wire#w7
   RUNG wire#powerrail
      { S7_Templates := "SrcType := Int" } GE_Contact(in1 := "BTrk".A0303.Stacker.Layers_Qty, in2 := "BTrk".A0303.Stacker.Layers_Target)
      wire#w8
      { S7_Templates := "SrcType := Int" } GT_Contact(in1 := "BTrk".A0303.Stacker.Layers_Target, in2 := 0)
      I_Contact( #Sts.Sollevatore.InPosPreDeposito )
      I_Contact( #CIn.Navetta.InPosizioneDiPrelievo )
      Coil( #Ctrl.Cycle.Sollevamento.PreDeposito )
      Move(in := 2, out1 => "A04_HMI".Synoptic.Impilatore.Fase)
   END_RUNG
   RUNG wire#powerrail
      Contact( "BTrk".A0303.Stacker.Completato )
   END_RUNG wire#w8
   RUNG wire#powerrail
      I_Contact( #Ctrl.Cycle.Sollevamento.Prelievo )
      I_Contact( #Ctrl.Cycle.Sollevamento.Deposito )
      I_Contact( #Ctrl.Cycle.Sollevamento.PreDeposito )
      Move(in := 0, out1 => "A04_HMI".Synoptic.Impilatore.Fase)
   END_RUNG
   // the same network as SCL:
   #Ctrl.Cycle.Sollevamento.Prelievo := ("BTrk".A0303.Stacker.Layers_Qty < "BTrk".A0303.Stacker.Layers_Target) AND NOT "BTrk".A0303.Stacker.Completato AND ((NOT #Sts.TraslazioneStrato.DropRequest AND NOT #Sts.Sollevatore.InPrePrelievoPos) OR (#Sts.TraslazioneStrato.DropRequest AND NOT #Sts.Sollevatore.InPrelievoPos)) AND NOT #Ctrl.Cycle.Sollevamento.Deposito AND ("BTrk".A0304.Empty OR (NOT "BTrk".A0304.Empty AND #CIn.Navetta.OutOfWorkspace)) AND (("BTrk".A0303.Transfert.Empty AND (#CIn.TraslazioneStrato.Ax_Testa.ActualPosition < (-700.0))) OR NOT "BTrk".A0303.Transfert.Empty);
   IF #Ctrl.Cycle.Sollevamento.Prelievo THEN "A04_HMI".Synoptic.Impilatore.Fase := 1; END_IF;
   #Ctrl.Cycle.Sollevamento.Deposito := #CIn.Navetta.InPosizioneDiPrelievo AND (("BTrk".A0303.Stacker.Layers_Qty >= "BTrk".A0303.Stacker.Layers_Target) OR "BTrk".A0303.Stacker.Completato) AND ("BTrk".A0303.Stacker.Layers_Target > 0) AND NOT #Sts.Sollevatore.InPosDeposito;
   IF #Ctrl.Cycle.Sollevamento.Deposito THEN "A04_HMI".Synoptic.Impilatore.Fase := 3; END_IF;
   #Ctrl.Cycle.Sollevamento.PreDeposito := (("BTrk".A0303.Stacker.Layers_Qty >= "BTrk".A0303.Stacker.Layers_Target) OR "BTrk".A0303.Stacker.Completato) AND ("BTrk".A0303.Stacker.Layers_Target > 0) AND NOT #Sts.Sollevatore.InPosPreDeposito AND NOT #CIn.Navetta.InPosizioneDiPrelievo;
   IF #Ctrl.Cycle.Sollevamento.PreDeposito THEN "A04_HMI".Synoptic.Impilatore.Fase := 2; END_IF;
   IF NOT #Ctrl.Cycle.Sollevamento.Prelievo AND NOT #Ctrl.Cycle.Sollevamento.Deposito AND NOT #Ctrl.Cycle.Sollevamento.PreDeposito THEN
       "A04_HMI".Synoptic.Impilatore.Fase := 0;
   END_IF;
END_REGION

REGION Network 45: Sollevatore Ready To Recive
   RUNG wire#powerrail
      Contact( #CIn.Sollevamento.Ax_Coda.Standstill )
      Contact( #CIn.Sollevamento.Ax_Testa.Standstill )
      Contact( #SollevatoreCodaInPrelievoPos )
      Contact( #SollevatoreTestaInPrelievoPos )
      { S7_Templates := "SrcType := Int" } LT_Contact(in1 := "BTrk".A0303.Stacker.Layers_Qty, in2 := "BTrk".A0303.Stacker.Layers_Target)
      I_Contact( "BTrk".A0303.Stacker.Completato )
      Coil( #Sts.Sollevatore.ReadyToRecive )
   END_RUNG
   // the same network as SCL:
   #Sts.Sollevatore.ReadyToRecive := #CIn.Sollevamento.Ax_Coda.Standstill AND #CIn.Sollevamento.Ax_Testa.Standstill AND #SollevatoreCodaInPrelievoPos AND #SollevatoreTestaInPrelievoPos AND ("BTrk".A0303.Stacker.Layers_Qty < "BTrk".A0303.Stacker.Layers_Target) AND NOT "BTrk".A0303.Stacker.Completato;
END_REGION

REGION Network 46: Sollevatore - COut Manager
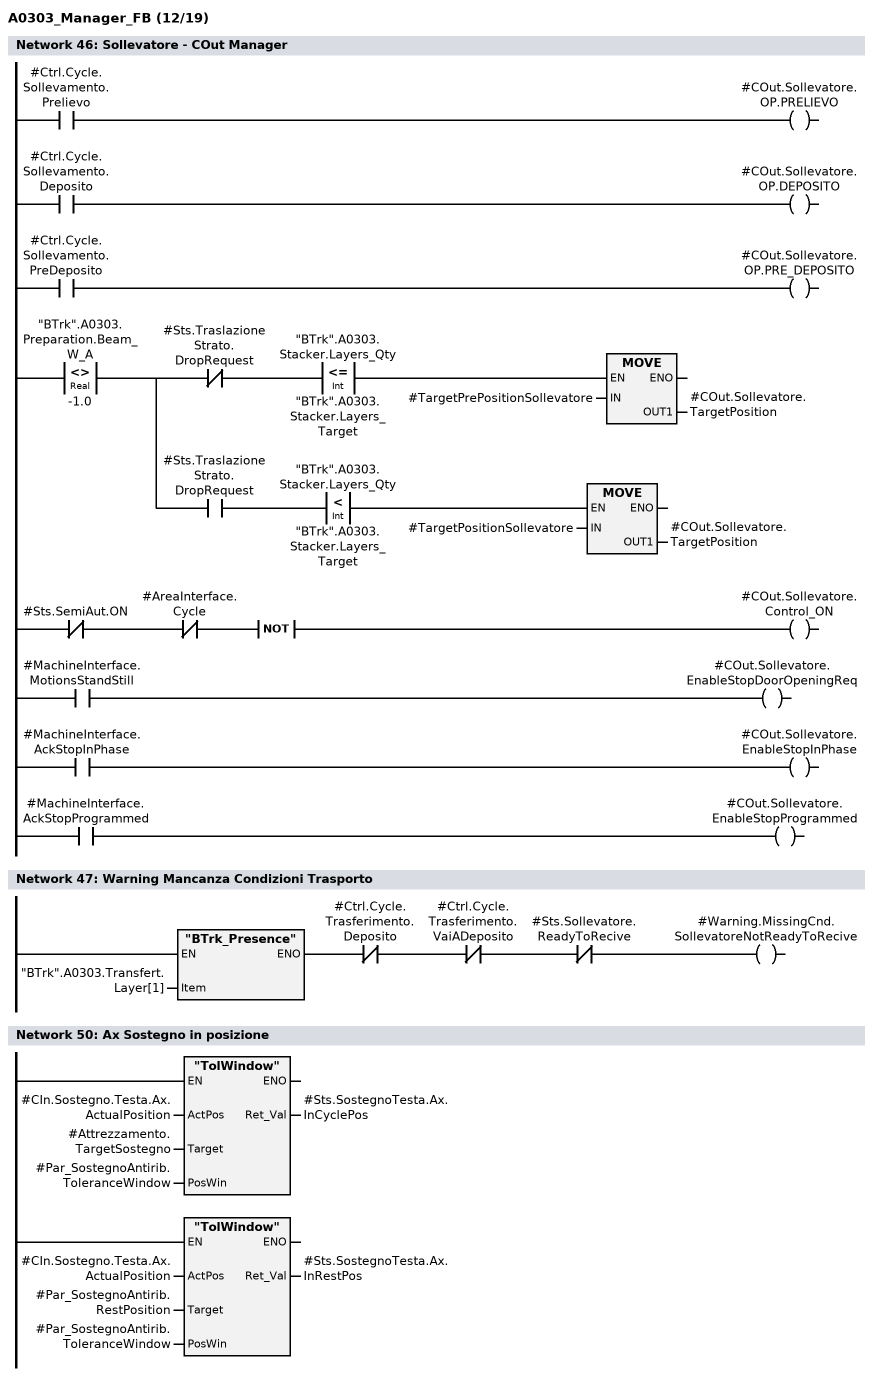
   RUNG wire#powerrail
      Contact( #Ctrl.Cycle.Sollevamento.Prelievo )
      Coil( #COut.Sollevatore.OP.PRELIEVO )
   END_RUNG
   RUNG wire#powerrail
      Contact( #Ctrl.Cycle.Sollevamento.Deposito )
      Coil( #COut.Sollevatore.OP.DEPOSITO )
   END_RUNG
   RUNG wire#powerrail
      Contact( #Ctrl.Cycle.Sollevamento.PreDeposito )
      Coil( #COut.Sollevatore.OP.PRE_DEPOSITO )
   END_RUNG
   RUNG wire#powerrail
      { S7_Templates := "SrcType := Real" } NE_Contact(in1 := "BTrk".A0303.Preparation.Beam_W_A, in2 := -1.0)
      wire#w1
      I_Contact( #Sts.TraslazioneStrato.DropRequest )
      { S7_Templates := "SrcType := Int" } LE_Contact(in1 := "BTrk".A0303.Stacker.Layers_Qty, in2 := "BTrk".A0303.Stacker.Layers_Target)
      Move(in := #TargetPrePositionSollevatore, out1 => #COut.Sollevatore.TargetPosition)
   END_RUNG
   RUNG wire#w1
      Contact( #Sts.TraslazioneStrato.DropRequest )
      { S7_Templates := "SrcType := Int" } LT_Contact(in1 := "BTrk".A0303.Stacker.Layers_Qty, in2 := "BTrk".A0303.Stacker.Layers_Target)
      Move(in := #TargetPositionSollevatore, out1 => #COut.Sollevatore.TargetPosition)
   END_RUNG
   RUNG wire#powerrail
      I_Contact( #Sts.SemiAut.ON )
      I_Contact( #AreaInterface.Cycle )
      Not()
      Coil( #COut.Sollevatore.Control_ON )
   END_RUNG
   RUNG wire#powerrail
      Contact( #MachineInterface.MotionsStandStill )
      Coil( #COut.Sollevatore.EnableStopDoorOpeningReq )
   END_RUNG
   RUNG wire#powerrail
      Contact( #MachineInterface.AckStopInPhase )
      Coil( #COut.Sollevatore.EnableStopInPhase )
   END_RUNG
   RUNG wire#powerrail
      Contact( #MachineInterface.AckStopProgrammed )
      Coil( #COut.Sollevatore.EnableStopProgrammed )
   END_RUNG
   // the same network as SCL:
   #COut.Sollevatore.OP.PRELIEVO := #Ctrl.Cycle.Sollevamento.Prelievo;
   #COut.Sollevatore.OP.DEPOSITO := #Ctrl.Cycle.Sollevamento.Deposito;
   #COut.Sollevatore.OP.PRE_DEPOSITO := #Ctrl.Cycle.Sollevamento.PreDeposito;
   #_w1 := "BTrk".A0303.Preparation.Beam_W_A <> (-1.0);
   IF #_w1 AND NOT #Sts.TraslazioneStrato.DropRequest AND ("BTrk".A0303.Stacker.Layers_Qty <= "BTrk".A0303.Stacker.Layers_Target) THEN
       #COut.Sollevatore.TargetPosition := #TargetPrePositionSollevatore;
   END_IF;
   IF #_w1 AND #Sts.TraslazioneStrato.DropRequest AND ("BTrk".A0303.Stacker.Layers_Qty < "BTrk".A0303.Stacker.Layers_Target) THEN
       #COut.Sollevatore.TargetPosition := #TargetPositionSollevatore;
   END_IF;
   #COut.Sollevatore.Control_ON := NOT (NOT #Sts.SemiAut.ON AND NOT #AreaInterface.Cycle);
   #COut.Sollevatore.EnableStopDoorOpeningReq := #MachineInterface.MotionsStandStill;
   #COut.Sollevatore.EnableStopInPhase := #MachineInterface.AckStopInPhase;
   #COut.Sollevatore.EnableStopProgrammed := #MachineInterface.AckStopProgrammed;
END_REGION

REGION Network 47: Warning Mancanza Condizioni Trasporto
   RUNG wire#powerrail
      "BTrk_Presence"(Item := "BTrk".A0303.Transfert.Layer[1])
      I_Contact( #Ctrl.Cycle.Trasferimento.Deposito )
      I_Contact( #Ctrl.Cycle.Trasferimento.VaiADeposito )
      I_Contact( #Sts.Sollevatore.ReadyToRecive )
      Coil( #Warning.MissingCnd.SollevatoreNotReadyToRecive )
   END_RUNG
   // the same network as SCL:
   "BTrk_Presence"(Item := "BTrk".A0303.Transfert.Layer[1], ENO => #_w1);
   #Warning.MissingCnd.SollevatoreNotReadyToRecive := #_w1 AND NOT #Ctrl.Cycle.Trasferimento.Deposito AND NOT #Ctrl.Cycle.Trasferimento.VaiADeposito AND NOT #Sts.Sollevatore.ReadyToRecive;
END_REGION

REGION Network 49: <<< SOSTEGNO TESTA >>>
END_REGION

REGION Network 50: Ax Sostegno in posizione
   RUNG wire#powerrail
      "TolWindow"(ActPos := #CIn.Sostegno.Testa.Ax.ActualPosition, Target := #Attrezzamento.TargetSostegno, PosWin := #Par_SostegnoAntirib.ToleranceWindow, Ret_Val => #Sts.SostegnoTesta.Ax.InCyclePos)
   END_RUNG
   RUNG wire#powerrail
      "TolWindow"(ActPos := #CIn.Sostegno.Testa.Ax.ActualPosition, Target := #Par_SostegnoAntirib.RestPosition, PosWin := #Par_SostegnoAntirib.ToleranceWindow, Ret_Val => #Sts.SostegnoTesta.Ax.InRestPos)
   END_RUNG
   // the same network as SCL:
   #Sts.SostegnoTesta.Ax.InCyclePos := "TolWindow"(ActPos := #CIn.Sostegno.Testa.Ax.ActualPosition,
                           Target := #Attrezzamento.TargetSostegno,
                           PosWin := #Par_SostegnoAntirib.ToleranceWindow);
   #Sts.SostegnoTesta.Ax.InRestPos := "TolWindow"(ActPos := #CIn.Sostegno.Testa.Ax.ActualPosition,
                           Target := #Par_SostegnoAntirib.RestPosition,
                           PosWin := #Par_SostegnoAntirib.ToleranceWindow);
END_REGION

REGION Network 51: Posizione PALETTI Antiribaltamento
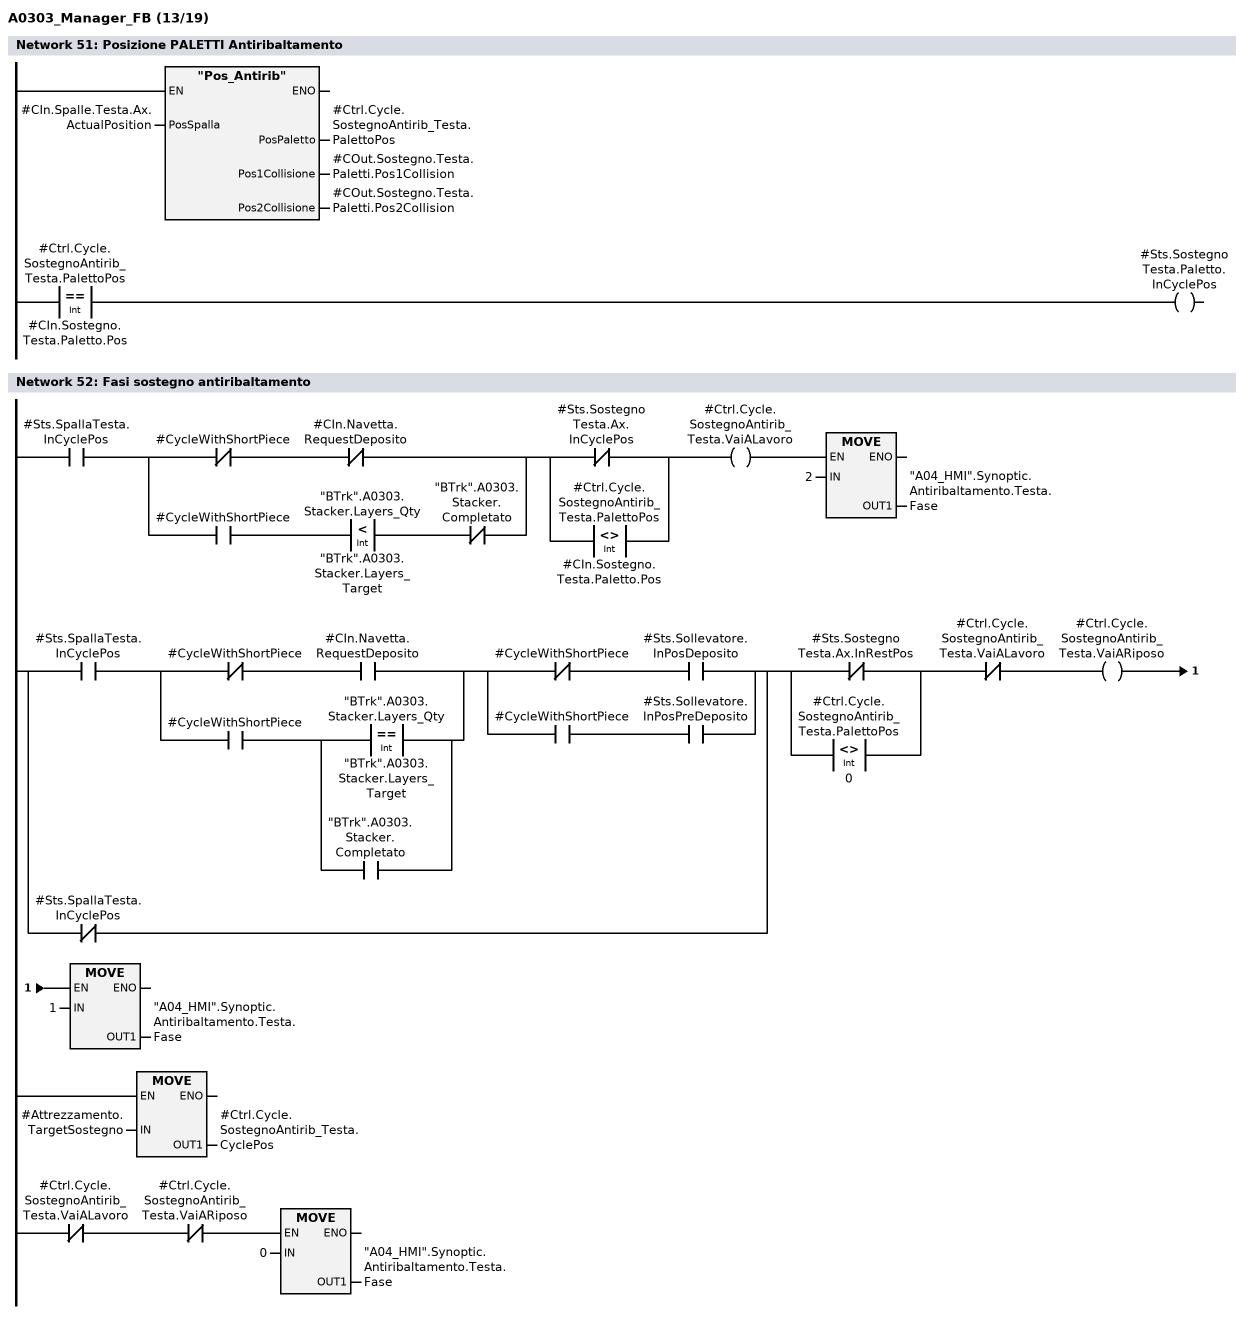
   RUNG wire#powerrail
      "Pos_Antirib"(PosSpalla := #CIn.Spalle.Testa.Ax.ActualPosition, PosPaletto => #Ctrl.Cycle.SostegnoAntirib_Testa.PalettoPos, Pos1Collisione => #COut.Sostegno.Testa.Paletti.Pos1Collision, Pos2Collisione => #COut.Sostegno.Testa.Paletti.Pos2Collision)
   END_RUNG
   RUNG wire#powerrail
      { S7_Templates := "SrcType := Int" } EQ_Contact(in1 := #Ctrl.Cycle.SostegnoAntirib_Testa.PalettoPos, in2 := #CIn.Sostegno.Testa.Paletto.Pos)
      Coil( #Sts.SostegnoTesta.Paletto.InCyclePos )
   END_RUNG
   // the same network as SCL:
   "Pos_Antirib"(PosSpalla := #CIn.Spalle.Testa.Ax.ActualPosition,
                 PosPaletto => #Ctrl.Cycle.SostegnoAntirib_Testa.PalettoPos,
                 Pos1Collisione => #COut.Sostegno.Testa.Paletti.Pos1Collision,
                 Pos2Collisione => #COut.Sostegno.Testa.Paletti.Pos2Collision);
   #Sts.SostegnoTesta.Paletto.InCyclePos := #Ctrl.Cycle.SostegnoAntirib_Testa.PalettoPos = #CIn.Sostegno.Testa.Paletto.Pos;
END_REGION

REGION Network 52: Fasi sostegno antiribaltamento
   RUNG wire#powerrail
      Contact( #Sts.SpallaTesta.InCyclePos )
      wire#w1
      I_Contact( #CycleWithShortPiece )
      I_Contact( #CIn.Navetta.RequestDeposito )
      wire#w2
      I_Contact( #Sts.SostegnoTesta.Ax.InCyclePos )
      wire#w3
      Coil( #Ctrl.Cycle.SostegnoAntirib_Testa.VaiALavoro )
      Move(in := 2, out1 => "A04_HMI".Synoptic.Antiribaltamento.Testa.Fase)
   END_RUNG
   RUNG wire#w1
      Contact( #CycleWithShortPiece )
      { S7_Templates := "SrcType := Int" } LT_Contact(in1 := "BTrk".A0303.Stacker.Layers_Qty, in2 := "BTrk".A0303.Stacker.Layers_Target)
      I_Contact( "BTrk".A0303.Stacker.Completato )
   END_RUNG wire#w2
   RUNG wire#w2
      { S7_Templates := "SrcType := Int" } NE_Contact(in1 := #Ctrl.Cycle.SostegnoAntirib_Testa.PalettoPos, in2 := #CIn.Sostegno.Testa.Paletto.Pos)
   END_RUNG wire#w3
   RUNG wire#powerrail
      Contact( #Sts.SpallaTesta.InCyclePos )
      wire#w4
      I_Contact( #CycleWithShortPiece )
      Contact( #CIn.Navetta.RequestDeposito )
      wire#w5
      I_Contact( #CycleWithShortPiece )
      Contact( #Sts.Sollevatore.InPosDeposito )
      wire#w7
      I_Contact( #Sts.SostegnoTesta.Ax.InRestPos )
      wire#w8
      I_Contact( #Ctrl.Cycle.SostegnoAntirib_Testa.VaiALavoro )
      Coil( #Ctrl.Cycle.SostegnoAntirib_Testa.VaiARiposo )
      Move(in := 1, out1 => "A04_HMI".Synoptic.Antiribaltamento.Testa.Fase)
   END_RUNG
   RUNG wire#w4
      Contact( #CycleWithShortPiece )
      wire#w6
      { S7_Templates := "SrcType := Int" } EQ_Contact(in1 := "BTrk".A0303.Stacker.Layers_Qty, in2 := "BTrk".A0303.Stacker.Layers_Target)
   END_RUNG wire#w5
   RUNG wire#w6
      Contact( "BTrk".A0303.Stacker.Completato )
   END_RUNG wire#w5
   RUNG wire#w5
      Contact( #CycleWithShortPiece )
      Contact( #Sts.Sollevatore.InPosPreDeposito )
   END_RUNG wire#w7
   RUNG wire#powerrail
      I_Contact( #Sts.SpallaTesta.InCyclePos )
   END_RUNG wire#w7
   RUNG wire#w7
      { S7_Templates := "SrcType := Int" } NE_Contact(in1 := #Ctrl.Cycle.SostegnoAntirib_Testa.PalettoPos, in2 := 0)
   END_RUNG wire#w8
   RUNG wire#powerrail
      Move(in := #Attrezzamento.TargetSostegno, out1 => #Ctrl.Cycle.SostegnoAntirib_Testa.CyclePos)
   END_RUNG
   RUNG wire#powerrail
      I_Contact( #Ctrl.Cycle.SostegnoAntirib_Testa.VaiALavoro )
      I_Contact( #Ctrl.Cycle.SostegnoAntirib_Testa.VaiARiposo )
      Move(in := 0, out1 => "A04_HMI".Synoptic.Antiribaltamento.Testa.Fase)
   END_RUNG
   // the same network as SCL:
   #Ctrl.Cycle.SostegnoAntirib_Testa.VaiALavoro := #Sts.SpallaTesta.InCyclePos AND ((NOT #CycleWithShortPiece AND NOT #CIn.Navetta.RequestDeposito) OR (#CycleWithShortPiece AND ("BTrk".A0303.Stacker.Layers_Qty < "BTrk".A0303.Stacker.Layers_Target) AND NOT "BTrk".A0303.Stacker.Completato)) AND (NOT #Sts.SostegnoTesta.Ax.InCyclePos OR (#Ctrl.Cycle.SostegnoAntirib_Testa.PalettoPos <> #CIn.Sostegno.Testa.Paletto.Pos));
   IF #Ctrl.Cycle.SostegnoAntirib_Testa.VaiALavoro THEN
       "A04_HMI".Synoptic.Antiribaltamento.Testa.Fase := 2;
   END_IF;
   #Ctrl.Cycle.SostegnoAntirib_Testa.VaiARiposo := ((#Sts.SpallaTesta.InCyclePos AND ((NOT #CycleWithShortPiece AND #CIn.Navetta.RequestDeposito) OR (#CycleWithShortPiece AND (("BTrk".A0303.Stacker.Layers_Qty = "BTrk".A0303.Stacker.Layers_Target) OR "BTrk".A0303.Stacker.Completato))) AND ((NOT #CycleWithShortPiece AND #Sts.Sollevatore.InPosDeposito) OR (#CycleWithShortPiece AND #Sts.Sollevatore.InPosPreDeposito))) OR NOT #Sts.SpallaTesta.InCyclePos) AND (NOT #Sts.SostegnoTesta.Ax.InRestPos OR (#Ctrl.Cycle.SostegnoAntirib_Testa.PalettoPos <> 0)) AND NOT #Ctrl.Cycle.SostegnoAntirib_Testa.VaiALavoro;
   IF #Ctrl.Cycle.SostegnoAntirib_Testa.VaiARiposo THEN
       "A04_HMI".Synoptic.Antiribaltamento.Testa.Fase := 1;
   END_IF;
   #Ctrl.Cycle.SostegnoAntirib_Testa.CyclePos := #Attrezzamento.TargetSostegno;
   IF NOT #Ctrl.Cycle.SostegnoAntirib_Testa.VaiALavoro AND NOT #Ctrl.Cycle.SostegnoAntirib_Testa.VaiARiposo THEN
       "A04_HMI".Synoptic.Antiribaltamento.Testa.Fase := 0;
   END_IF;
END_REGION

REGION Network 53: Sostegno Testa - COut Manager
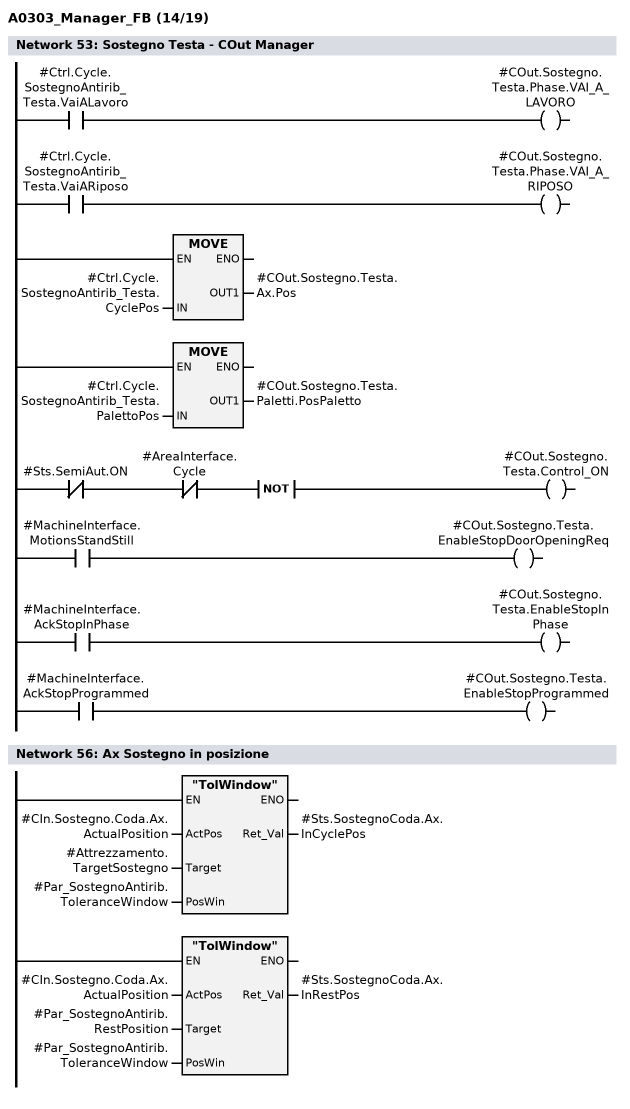
   RUNG wire#powerrail
      Contact( #Ctrl.Cycle.SostegnoAntirib_Testa.VaiALavoro )
      Coil( #COut.Sostegno.Testa.Phase.VAI_A_LAVORO )
   END_RUNG
   RUNG wire#powerrail
      Contact( #Ctrl.Cycle.SostegnoAntirib_Testa.VaiARiposo )
      Coil( #COut.Sostegno.Testa.Phase.VAI_A_RIPOSO )
   END_RUNG
   RUNG wire#powerrail
      Move(in := #Ctrl.Cycle.SostegnoAntirib_Testa.CyclePos, out1 => #COut.Sostegno.Testa.Ax.Pos)
   END_RUNG
   RUNG wire#powerrail
      Move(in := #Ctrl.Cycle.SostegnoAntirib_Testa.PalettoPos, out1 => #COut.Sostegno.Testa.Paletti.PosPaletto)
   END_RUNG
   RUNG wire#powerrail
      I_Contact( #Sts.SemiAut.ON )
      I_Contact( #AreaInterface.Cycle )
      Not()
      Coil( #COut.Sostegno.Testa.Control_ON )
   END_RUNG
   RUNG wire#powerrail
      Contact( #MachineInterface.MotionsStandStill )
      Coil( #COut.Sostegno.Testa.EnableStopDoorOpeningReq )
   END_RUNG
   RUNG wire#powerrail
      Contact( #MachineInterface.AckStopInPhase )
      Coil( #COut.Sostegno.Testa.EnableStopInPhase )
   END_RUNG
   RUNG wire#powerrail
      Contact( #MachineInterface.AckStopProgrammed )
      Coil( #COut.Sostegno.Testa.EnableStopProgrammed )
   END_RUNG
   // the same network as SCL:
   #COut.Sostegno.Testa.Phase.VAI_A_LAVORO := #Ctrl.Cycle.SostegnoAntirib_Testa.VaiALavoro;
   #COut.Sostegno.Testa.Phase.VAI_A_RIPOSO := #Ctrl.Cycle.SostegnoAntirib_Testa.VaiARiposo;
   #COut.Sostegno.Testa.Ax.Pos := #Ctrl.Cycle.SostegnoAntirib_Testa.CyclePos;
   #COut.Sostegno.Testa.Paletti.PosPaletto := #Ctrl.Cycle.SostegnoAntirib_Testa.PalettoPos;
   #COut.Sostegno.Testa.Control_ON := NOT (NOT #Sts.SemiAut.ON AND NOT #AreaInterface.Cycle);
   #COut.Sostegno.Testa.EnableStopDoorOpeningReq := #MachineInterface.MotionsStandStill;
   #COut.Sostegno.Testa.EnableStopInPhase := #MachineInterface.AckStopInPhase;
   #COut.Sostegno.Testa.EnableStopProgrammed := #MachineInterface.AckStopProgrammed;
END_REGION

REGION Network 55: <<< SOSTEGNO CODA >>>
END_REGION

REGION Network 56: Ax Sostegno in posizione
   RUNG wire#powerrail
      "TolWindow"(ActPos := #CIn.Sostegno.Coda.Ax.ActualPosition, Target := #Attrezzamento.TargetSostegno, PosWin := #Par_SostegnoAntirib.ToleranceWindow, Ret_Val => #Sts.SostegnoCoda.Ax.InCyclePos)
   END_RUNG
   RUNG wire#powerrail
      "TolWindow"(ActPos := #CIn.Sostegno.Coda.Ax.ActualPosition, Target := #Par_SostegnoAntirib.RestPosition, PosWin := #Par_SostegnoAntirib.ToleranceWindow, Ret_Val => #Sts.SostegnoCoda.Ax.InRestPos)
   END_RUNG
   // the same network as SCL:
   #Sts.SostegnoCoda.Ax.InCyclePos := "TolWindow"(ActPos := #CIn.Sostegno.Coda.Ax.ActualPosition,
                           Target := #Attrezzamento.TargetSostegno,
                           PosWin := #Par_SostegnoAntirib.ToleranceWindow);
   #Sts.SostegnoCoda.Ax.InRestPos := "TolWindow"(ActPos := #CIn.Sostegno.Coda.Ax.ActualPosition,
                           Target := #Par_SostegnoAntirib.RestPosition,
                           PosWin := #Par_SostegnoAntirib.ToleranceWindow);
END_REGION

REGION Network 57: Posizione PALETTI Antiribaltamento
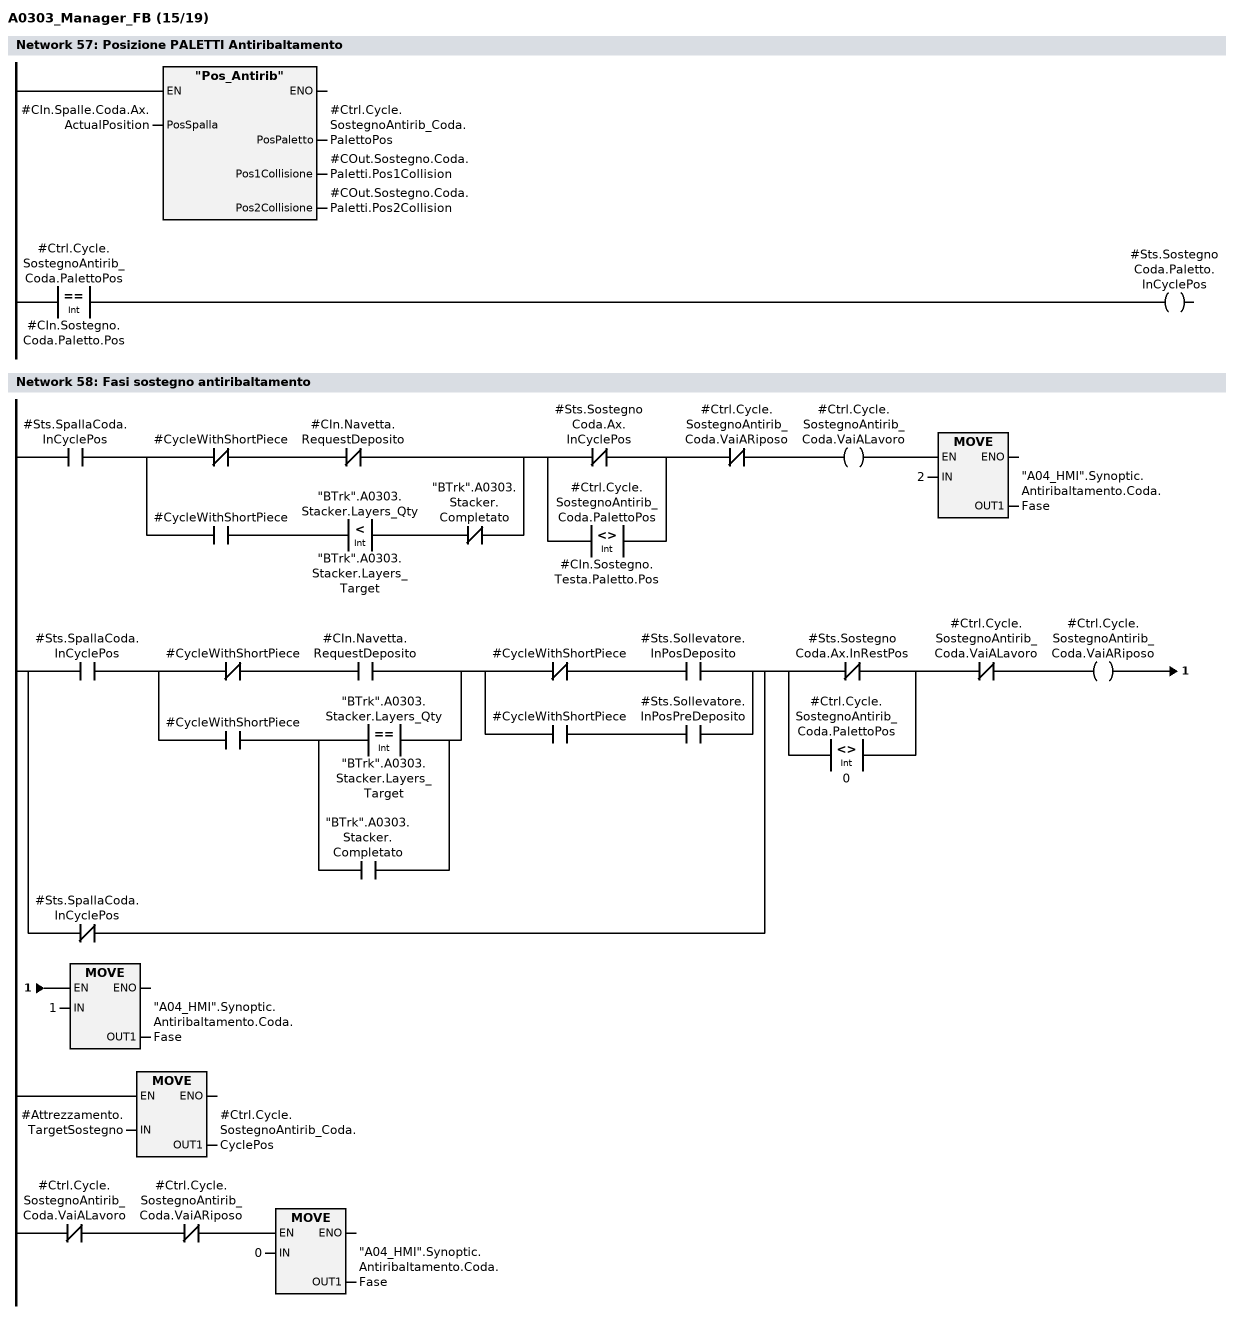
   RUNG wire#powerrail
      "Pos_Antirib"(PosSpalla := #CIn.Spalle.Coda.Ax.ActualPosition, PosPaletto => #Ctrl.Cycle.SostegnoAntirib_Coda.PalettoPos, Pos1Collisione => #COut.Sostegno.Coda.Paletti.Pos1Collision, Pos2Collisione => #COut.Sostegno.Coda.Paletti.Pos2Collision)
   END_RUNG
   RUNG wire#powerrail
      { S7_Templates := "SrcType := Int" } EQ_Contact(in1 := #Ctrl.Cycle.SostegnoAntirib_Coda.PalettoPos, in2 := #CIn.Sostegno.Coda.Paletto.Pos)
      Coil( #Sts.SostegnoCoda.Paletto.InCyclePos )
   END_RUNG
   // the same network as SCL:
   "Pos_Antirib"(PosSpalla := #CIn.Spalle.Coda.Ax.ActualPosition,
                 PosPaletto => #Ctrl.Cycle.SostegnoAntirib_Coda.PalettoPos,
                 Pos1Collisione => #COut.Sostegno.Coda.Paletti.Pos1Collision,
                 Pos2Collisione => #COut.Sostegno.Coda.Paletti.Pos2Collision);
   #Sts.SostegnoCoda.Paletto.InCyclePos := #Ctrl.Cycle.SostegnoAntirib_Coda.PalettoPos = #CIn.Sostegno.Coda.Paletto.Pos;
END_REGION

REGION Network 58: Fasi sostegno antiribaltamento
   RUNG wire#powerrail
      Contact( #Sts.SpallaCoda.InCyclePos )
      wire#w1
      I_Contact( #CycleWithShortPiece )
      I_Contact( #CIn.Navetta.RequestDeposito )
      wire#w2
      I_Contact( #Sts.SostegnoCoda.Ax.InCyclePos )
      wire#w3
      I_Contact( #Ctrl.Cycle.SostegnoAntirib_Coda.VaiARiposo )
      Coil( #Ctrl.Cycle.SostegnoAntirib_Coda.VaiALavoro )
      Move(in := 2, out1 => "A04_HMI".Synoptic.Antiribaltamento.Coda.Fase)
   END_RUNG
   RUNG wire#w1
      Contact( #CycleWithShortPiece )
      { S7_Templates := "SrcType := Int" } LT_Contact(in1 := "BTrk".A0303.Stacker.Layers_Qty, in2 := "BTrk".A0303.Stacker.Layers_Target)
      I_Contact( "BTrk".A0303.Stacker.Completato )
   END_RUNG wire#w2
   RUNG wire#w2
      { S7_Templates := "SrcType := Int" } NE_Contact(in1 := #Ctrl.Cycle.SostegnoAntirib_Coda.PalettoPos, in2 := #CIn.Sostegno.Testa.Paletto.Pos)
   END_RUNG wire#w3
   RUNG wire#powerrail
      Contact( #Sts.SpallaCoda.InCyclePos )
      wire#w4
      I_Contact( #CycleWithShortPiece )
      Contact( #CIn.Navetta.RequestDeposito )
      wire#w5
      I_Contact( #CycleWithShortPiece )
      Contact( #Sts.Sollevatore.InPosDeposito )
      wire#w7
      I_Contact( #Sts.SostegnoCoda.Ax.InRestPos )
      wire#w8
      I_Contact( #Ctrl.Cycle.SostegnoAntirib_Coda.VaiALavoro )
      Coil( #Ctrl.Cycle.SostegnoAntirib_Coda.VaiARiposo )
      Move(in := 1, out1 => "A04_HMI".Synoptic.Antiribaltamento.Coda.Fase)
   END_RUNG
   RUNG wire#w4
      Contact( #CycleWithShortPiece )
      wire#w6
      { S7_Templates := "SrcType := Int" } EQ_Contact(in1 := "BTrk".A0303.Stacker.Layers_Qty, in2 := "BTrk".A0303.Stacker.Layers_Target)
   END_RUNG wire#w5
   RUNG wire#w6
      Contact( "BTrk".A0303.Stacker.Completato )
   END_RUNG wire#w5
   RUNG wire#w5
      Contact( #CycleWithShortPiece )
      Contact( #Sts.Sollevatore.InPosPreDeposito )
   END_RUNG wire#w7
   RUNG wire#powerrail
      I_Contact( #Sts.SpallaCoda.InCyclePos )
   END_RUNG wire#w7
   RUNG wire#w7
      { S7_Templates := "SrcType := Int" } NE_Contact(in1 := #Ctrl.Cycle.SostegnoAntirib_Coda.PalettoPos, in2 := 0)
   END_RUNG wire#w8
   RUNG wire#powerrail
      Move(in := #Attrezzamento.TargetSostegno, out1 => #Ctrl.Cycle.SostegnoAntirib_Coda.CyclePos)
   END_RUNG
   RUNG wire#powerrail
      I_Contact( #Ctrl.Cycle.SostegnoAntirib_Coda.VaiALavoro )
      I_Contact( #Ctrl.Cycle.SostegnoAntirib_Coda.VaiARiposo )
      Move(in := 0, out1 => "A04_HMI".Synoptic.Antiribaltamento.Coda.Fase)
   END_RUNG
   // the same network as SCL:
   #Ctrl.Cycle.SostegnoAntirib_Coda.VaiALavoro := #Sts.SpallaCoda.InCyclePos AND ((NOT #CycleWithShortPiece AND NOT #CIn.Navetta.RequestDeposito) OR (#CycleWithShortPiece AND ("BTrk".A0303.Stacker.Layers_Qty < "BTrk".A0303.Stacker.Layers_Target) AND NOT "BTrk".A0303.Stacker.Completato)) AND (NOT #Sts.SostegnoCoda.Ax.InCyclePos OR (#Ctrl.Cycle.SostegnoAntirib_Coda.PalettoPos <> #CIn.Sostegno.Testa.Paletto.Pos)) AND NOT #Ctrl.Cycle.SostegnoAntirib_Coda.VaiARiposo;
   IF #Ctrl.Cycle.SostegnoAntirib_Coda.VaiALavoro THEN
       "A04_HMI".Synoptic.Antiribaltamento.Coda.Fase := 2;
   END_IF;
   #Ctrl.Cycle.SostegnoAntirib_Coda.VaiARiposo := ((#Sts.SpallaCoda.InCyclePos AND ((NOT #CycleWithShortPiece AND #CIn.Navetta.RequestDeposito) OR (#CycleWithShortPiece AND (("BTrk".A0303.Stacker.Layers_Qty = "BTrk".A0303.Stacker.Layers_Target) OR "BTrk".A0303.Stacker.Completato))) AND ((NOT #CycleWithShortPiece AND #Sts.Sollevatore.InPosDeposito) OR (#CycleWithShortPiece AND #Sts.Sollevatore.InPosPreDeposito))) OR NOT #Sts.SpallaCoda.InCyclePos) AND (NOT #Sts.SostegnoCoda.Ax.InRestPos OR (#Ctrl.Cycle.SostegnoAntirib_Coda.PalettoPos <> 0)) AND NOT #Ctrl.Cycle.SostegnoAntirib_Coda.VaiALavoro;
   IF #Ctrl.Cycle.SostegnoAntirib_Coda.VaiARiposo THEN
       "A04_HMI".Synoptic.Antiribaltamento.Coda.Fase := 1;
   END_IF;
   #Ctrl.Cycle.SostegnoAntirib_Coda.CyclePos := #Attrezzamento.TargetSostegno;
   IF NOT #Ctrl.Cycle.SostegnoAntirib_Coda.VaiALavoro AND NOT #Ctrl.Cycle.SostegnoAntirib_Coda.VaiARiposo THEN
       "A04_HMI".Synoptic.Antiribaltamento.Coda.Fase := 0;
   END_IF;
END_REGION

REGION Network 59: Sostegno Coda - COut Manager
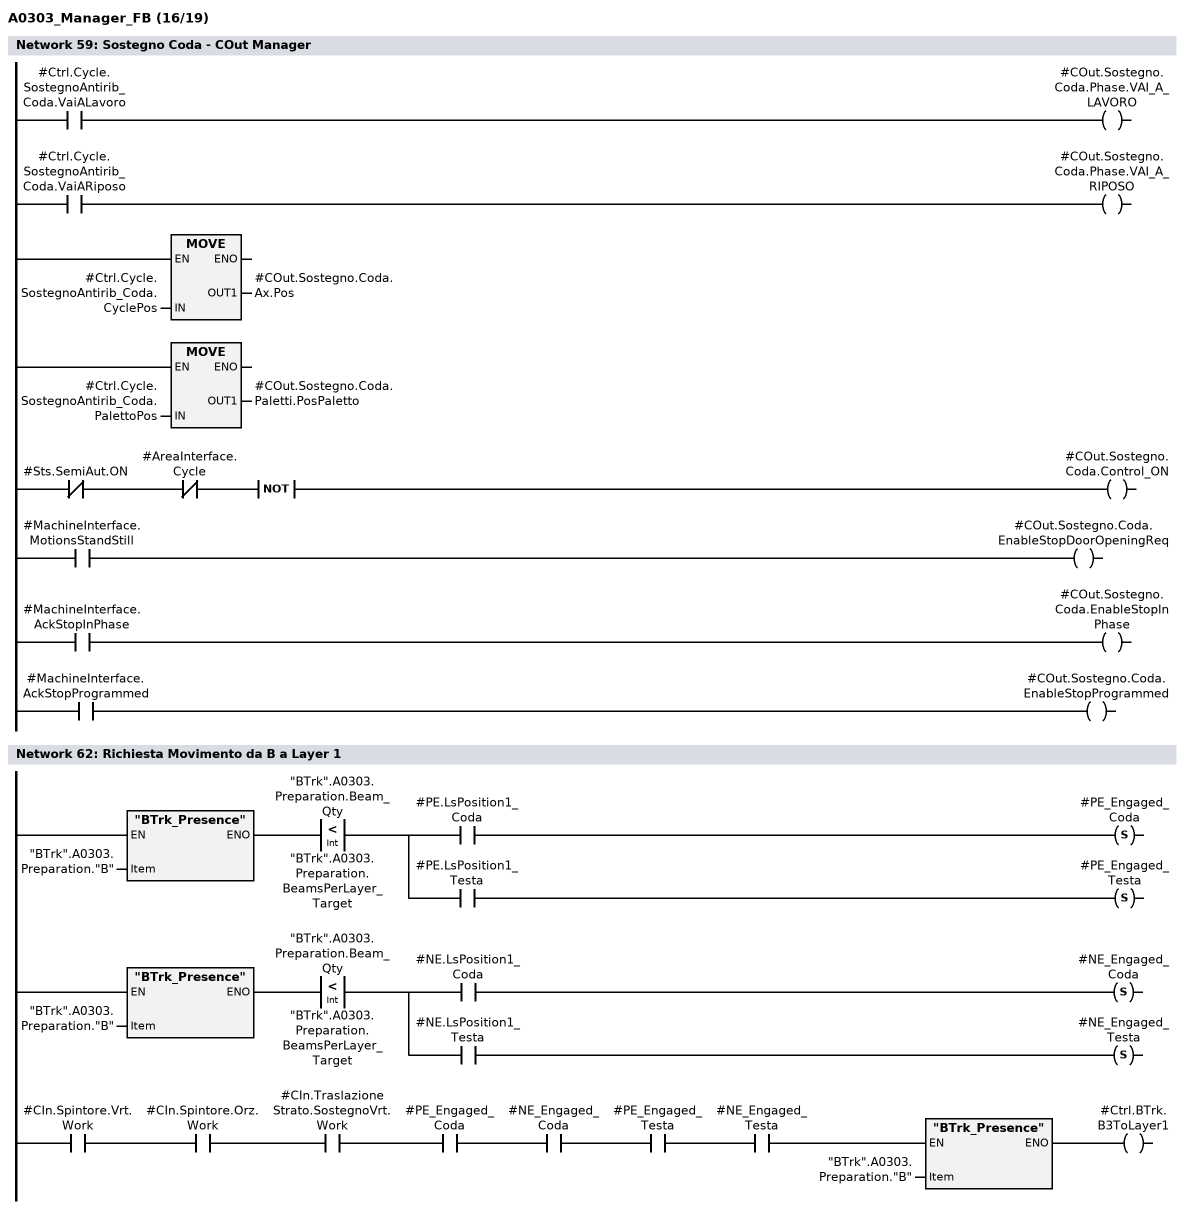
   RUNG wire#powerrail
      Contact( #Ctrl.Cycle.SostegnoAntirib_Coda.VaiALavoro )
      Coil( #COut.Sostegno.Coda.Phase.VAI_A_LAVORO )
   END_RUNG
   RUNG wire#powerrail
      Contact( #Ctrl.Cycle.SostegnoAntirib_Coda.VaiARiposo )
      Coil( #COut.Sostegno.Coda.Phase.VAI_A_RIPOSO )
   END_RUNG
   RUNG wire#powerrail
      Move(in := #Ctrl.Cycle.SostegnoAntirib_Coda.CyclePos, out1 => #COut.Sostegno.Coda.Ax.Pos)
   END_RUNG
   RUNG wire#powerrail
      Move(in := #Ctrl.Cycle.SostegnoAntirib_Coda.PalettoPos, out1 => #COut.Sostegno.Coda.Paletti.PosPaletto)
   END_RUNG
   RUNG wire#powerrail
      I_Contact( #Sts.SemiAut.ON )
      I_Contact( #AreaInterface.Cycle )
      Not()
      Coil( #COut.Sostegno.Coda.Control_ON )
   END_RUNG
   RUNG wire#powerrail
      Contact( #MachineInterface.MotionsStandStill )
      Coil( #COut.Sostegno.Coda.EnableStopDoorOpeningReq )
   END_RUNG
   RUNG wire#powerrail
      Contact( #MachineInterface.AckStopInPhase )
      Coil( #COut.Sostegno.Coda.EnableStopInPhase )
   END_RUNG
   RUNG wire#powerrail
      Contact( #MachineInterface.AckStopProgrammed )
      Coil( #COut.Sostegno.Coda.EnableStopProgrammed )
   END_RUNG
   // the same network as SCL:
   #COut.Sostegno.Coda.Phase.VAI_A_LAVORO := #Ctrl.Cycle.SostegnoAntirib_Coda.VaiALavoro;
   #COut.Sostegno.Coda.Phase.VAI_A_RIPOSO := #Ctrl.Cycle.SostegnoAntirib_Coda.VaiARiposo;
   #COut.Sostegno.Coda.Ax.Pos := #Ctrl.Cycle.SostegnoAntirib_Coda.CyclePos;
   #COut.Sostegno.Coda.Paletti.PosPaletto := #Ctrl.Cycle.SostegnoAntirib_Coda.PalettoPos;
   #COut.Sostegno.Coda.Control_ON := NOT (NOT #Sts.SemiAut.ON AND NOT #AreaInterface.Cycle);
   #COut.Sostegno.Coda.EnableStopDoorOpeningReq := #MachineInterface.MotionsStandStill;
   #COut.Sostegno.Coda.EnableStopInPhase := #MachineInterface.AckStopInPhase;
   #COut.Sostegno.Coda.EnableStopProgrammed := #MachineInterface.AckStopProgrammed;
END_REGION

REGION Network 61: <<<<<<<<<<<< MOVIMENTAZIONE TRACKING>>>>>>>>>>>>>>
END_REGION

REGION Network 62: Richiesta Movimento da B a Layer 1
   RUNG wire#powerrail
      "BTrk_Presence"(Item := "BTrk".A0303.Preparation."B")
      { S7_Templates := "SrcType := Int" } LT_Contact(in1 := "BTrk".A0303.Preparation.Beam_Qty, in2 := "BTrk".A0303.Preparation.BeamsPerLayer_Target)
      wire#w1
      Contact( #PE.LsPosition1_Coda )
      S_Coil( #PE_Engaged_Coda )
   END_RUNG
   RUNG wire#w1
      Contact( #PE.LsPosition1_Testa )
      S_Coil( #PE_Engaged_Testa )
   END_RUNG
   RUNG wire#powerrail
      "BTrk_Presence"(Item := "BTrk".A0303.Preparation."B")
      { S7_Templates := "SrcType := Int" } LT_Contact(in1 := "BTrk".A0303.Preparation.Beam_Qty, in2 := "BTrk".A0303.Preparation.BeamsPerLayer_Target)
      wire#w2
      Contact( #NE.LsPosition1_Coda )
      S_Coil( #NE_Engaged_Coda )
   END_RUNG
   RUNG wire#w2
      Contact( #NE.LsPosition1_Testa )
      S_Coil( #NE_Engaged_Testa )
   END_RUNG
   RUNG wire#powerrail
      Contact( #CIn.Spintore.Vrt.Work )
      Contact( #CIn.Spintore.Orz.Work )
      Contact( #CIn.TraslazioneStrato.SostegnoVrt.Work )
      Contact( #PE_Engaged_Coda )
      Contact( #NE_Engaged_Coda )
      Contact( #PE_Engaged_Testa )
      Contact( #NE_Engaged_Testa )
      "BTrk_Presence"(Item := "BTrk".A0303.Preparation."B")
      Coil( #Ctrl.BTrk.B3ToLayer1 )
   END_RUNG
   // the same network as SCL:
   "BTrk_Presence"(Item := "BTrk".A0303.Preparation."B", ENO => #_w1);
   #_w2 := #_w1 AND ("BTrk".A0303.Preparation.Beam_Qty < "BTrk".A0303.Preparation.BeamsPerLayer_Target);
   IF #_w2 AND #PE.LsPosition1_Coda THEN #PE_Engaged_Coda := TRUE; END_IF;
   IF #_w2 AND #PE.LsPosition1_Testa THEN #PE_Engaged_Testa := TRUE; END_IF;
   "BTrk_Presence"(Item := "BTrk".A0303.Preparation."B", ENO => #_w3);
   #_w4 := #_w3 AND ("BTrk".A0303.Preparation.Beam_Qty < "BTrk".A0303.Preparation.BeamsPerLayer_Target);
   IF #_w4 AND #NE.LsPosition1_Coda THEN #NE_Engaged_Coda := TRUE; END_IF;
   IF #_w4 AND #NE.LsPosition1_Testa THEN #NE_Engaged_Testa := TRUE; END_IF;
   "BTrk_Presence"(EN := #CIn.Spintore.Vrt.Work AND #CIn.Spintore.Orz.Work AND #CIn.TraslazioneStrato.SostegnoVrt.Work AND #PE_Engaged_Coda AND #NE_Engaged_Coda AND #PE_Engaged_Testa AND #NE_Engaged_Testa,
                   Item := "BTrk".A0303.Preparation."B",
                   ENO => #_w5);
   #Ctrl.BTrk.B3ToLayer1 := #_w5;
END_REGION

REGION Network 64 (SCL): Movimento BTRK da B0 == a ==> Layer 1 + shift a destra dei layer
   IF "BTrk".A0303.Preparation.BeamsPerLayer_Target <> 0 THEN

       IF #Ctrl.BTrk.B3ToLayer1 THEN

           IF "BTrk".A0303.Preparation.Beam_Qty < "BTrk".A0303.Preparation.BeamsPerLayer_Target THEN

               //Controllo che non sia gia pieno altrimenti allarme
               //
               IF "BTrk".A0303.Preparation.Beam_Qty > 0 THEN
                   // Cerco se ci sono degli spazi vuoti dovuti da un delete del trk manuale
                   // 
                   FOR #i := 1 TO "BTrk".A0303.Preparation.Beam_Qty  DO
                       IF "BTrk".A0303.Preparation.Layer[#i].B_ID = 0 THEN
                           #EmptyNFound := #i;
                           EXIT;
                       END_IF;
                       #EmptyNFound := 0;

                   END_FOR;
               END_IF;
               IF #EmptyNFound > 0 THEN
                   #ShiftN := #EmptyNFound;
               ELSE
                   #ShiftN := "BTrk".A0303.Preparation.BeamsPerLayer_Target;
               END_IF;


               #ShiftArrayOk := MOVE_BLK_VARIANT(
                                           SRC := "BTrk".A0303.Preparation.Layer,
                                           COUNT := #ShiftN - 1,// numero di elementi da spostare
                                           SRC_INDEX := 0,
                                           DEST_INDEX := 1,
                                           DEST => "BTrk".A0303.Preparation.Layer);



               // Inserimento nuovo valore nel primo layer
               "BTrk".A0303.Preparation.Layer[1] := "BTrk".A0303.Preparation.B;

               // Svuotamento B2
               "BTrk".A0303.Preparation.B := "BTrk".Empty;

           ELSE
               #Alarm.TrkPreparationAlreadyFull := TRUE;

           END_IF;
           #PE_Engaged_Coda := FALSE;
           #NE_Engaged_Coda := FALSE;
           #PE_Engaged_Testa := FALSE;
           #NE_Engaged_Testa := FALSE;


       END_IF;
   END_IF;
END_REGION

REGION Network 65 (SCL): Pacco Preparation completato / vuoto / conteggio pezzi
   // Conteggio Pezzi
   #ConteggioPezzi_Preparation := 0;
   FOR #i := 1 TO "BTrk".A0303.Preparation.BeamsPerLayer_Target DO
       IF "BTrk".A0303.Preparation.Layer[#i].B_ID > 0 THEN
           #ConteggioPezzi_Preparation += 1;
       END_IF;
   END_FOR;

   "BTrk".A0303.Preparation.Beam_Qty := #ConteggioPezzi_Preparation;

   // pallet empty/full
   "BTrk".A0303.Preparation.Empty := #ConteggioPezzi_Preparation = 0;

   IF "BTrk".A0303.Preparation.Empty THEN
       "BTrk".A0303.Preparation.Completato := FALSE;
   END_IF;
END_REGION

REGION Network 66: Tracking from Preparation to Transfer
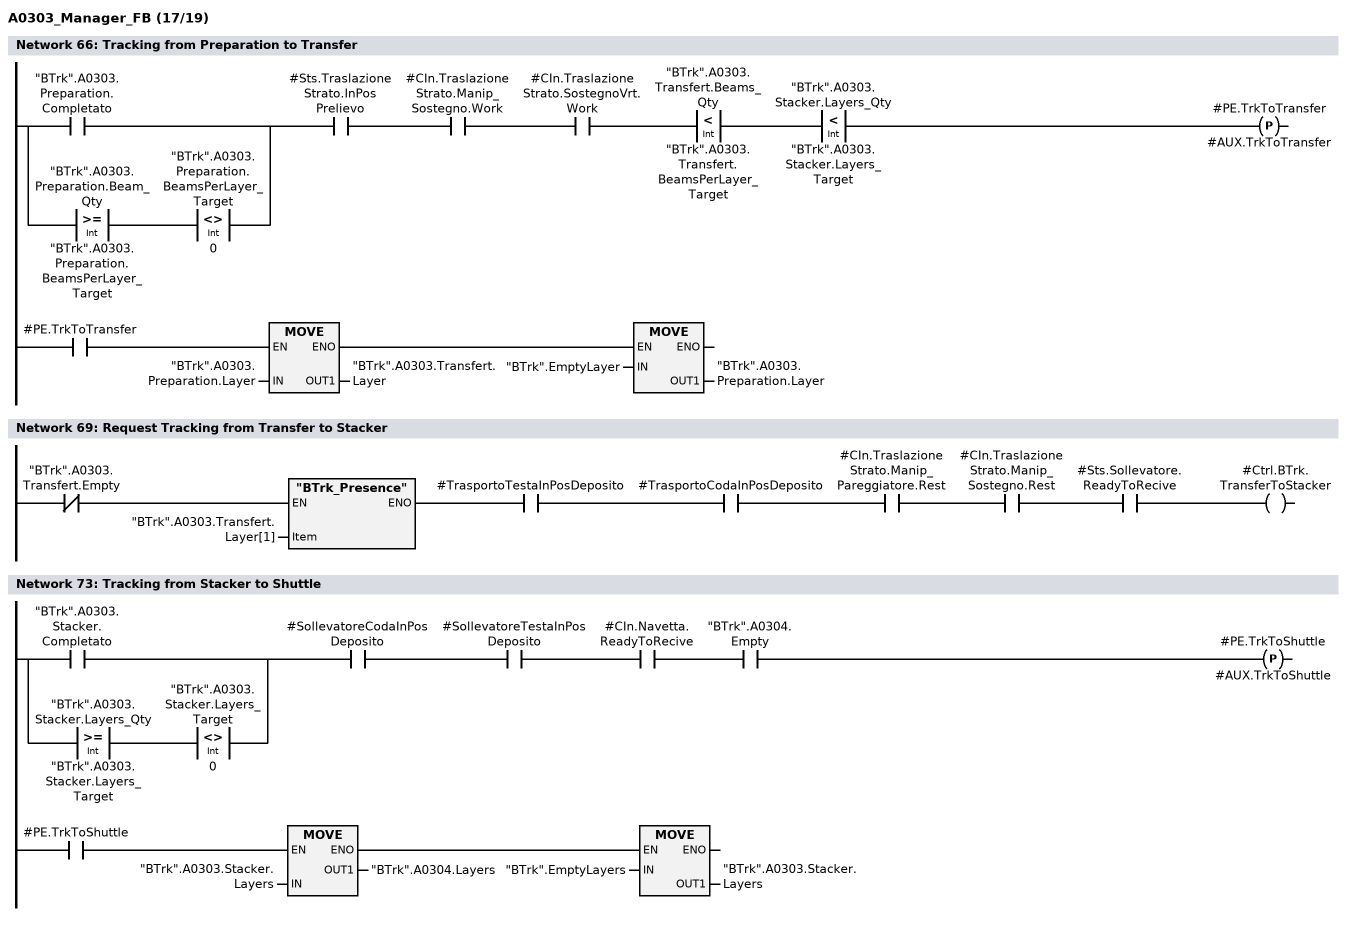
   #_w1 := ("BTrk".A0303.Preparation.Completato OR (("BTrk".A0303.Preparation.Beam_Qty >= "BTrk".A0303.Preparation.BeamsPerLayer_Target) AND ("BTrk".A0303.Preparation.BeamsPerLayer_Target <> 0))) AND #Sts.TraslazioneStrato.InPosPrelievo AND #CIn.TraslazioneStrato.Manip_Sostegno.Work AND #CIn.TraslazioneStrato.SostegnoVrt.Work AND ("BTrk".A0303.Transfert.Beams_Qty < "BTrk".A0303.Transfert.BeamsPerLayer_Target) AND ("BTrk".A0303.Stacker.Layers_Qty < "BTrk".A0303.Stacker.Layers_Target);
   #PE.TrkToTransfer := #_w1 AND NOT #AUX.TrkToTransfer;   // rising edge
   #AUX.TrkToTransfer := #_w1;
   IF #PE.TrkToTransfer THEN
       "BTrk".A0303.Transfert.Layer := "BTrk".A0303.Preparation.Layer;
       "BTrk".A0303.Preparation.Layer := "BTrk".EmptyLayer;
   END_IF;
END_REGION

REGION Network 67 (SCL): Transfert vuoto / conteggio pezzi
   // Conteggio Pezzi
   #ConteggioPezzi_Transfert := 0;
   FOR #i := 1 TO "BTrk".A0303.Transfert.BeamsPerLayer_Target DO
       IF  "BTrk".A0303.Transfert.Layer[#i].B_ID> 0 THEN
           #ConteggioPezzi_Transfert += 1;
       END_IF;
   END_FOR;

   "BTrk".A0303.Transfert.Beams_Qty:= #ConteggioPezzi_Transfert;

   // pallet empty/full
   "BTrk".A0303.Transfert.Empty := #ConteggioPezzi_Transfert = 0;
END_REGION

REGION Network 69: Request Tracking from Transfer to Stacker
   RUNG wire#powerrail
      I_Contact( "BTrk".A0303.Transfert.Empty )
      "BTrk_Presence"(Item := "BTrk".A0303.Transfert.Layer[1])
      Contact( #TrasportoTestaInPosDeposito )
      Contact( #TrasportoCodaInPosDeposito )
      Contact( #CIn.TraslazioneStrato.Manip_Pareggiatore.Rest )
      Contact( #CIn.TraslazioneStrato.Manip_Sostegno.Rest )
      Contact( #Sts.Sollevatore.ReadyToRecive )
      Coil( #Ctrl.BTrk.TransferToStacker )
   END_RUNG
   // the same network as SCL:
   "BTrk_Presence"(EN := NOT "BTrk".A0303.Transfert.Empty, Item := "BTrk".A0303.Transfert.Layer[1], ENO => #_w1);
   #Ctrl.BTrk.TransferToStacker := #_w1 AND #TrasportoTestaInPosDeposito AND #TrasportoCodaInPosDeposito AND #CIn.TraslazioneStrato.Manip_Pareggiatore.Rest AND #CIn.TraslazioneStrato.Manip_Sostegno.Rest AND #Sts.Sollevatore.ReadyToRecive;
END_REGION

REGION Network 70 (SCL): Pacco Stacker completato / vuoto / conteggio pezzi
   // Conteggio Pezzi
   #ConteggioPezzi_Stacker := 0;
   FOR #i := 1 TO "BTrk".A0303.Stacker.Layers_Target DO
       IF  "BTrk".A0303.Stacker.Layers[#i].Layer[1].B_ID> 0 THEN
           #ConteggioPezzi_Stacker += 1;
       END_IF;
   END_FOR;

   "BTrk".A0303.Stacker.Layers_Qty:= #ConteggioPezzi_Stacker;

   // pallet empty/full
   "BTrk".A0303.Stacker.Empty := #ConteggioPezzi_Stacker = 0;

   IF "BTrk".A0303.Stacker.Empty THEN
       "BTrk".A0303.Stacker.Completato := FALSE;
   END_IF;
END_REGION

REGION Network 71 (SCL): Tracking from Transfer to Stacker
   // Metto sempre l'ultimo strato depositato nel Layer 1 e shifto a destra gli altri elementi
   IF #Ctrl.BTrk.TransferToStacker THEN

       IF "BTrk".A0303.Stacker.Layers_Qty < "BTrk".A0303.Stacker.Layers_Target THEN  //Controllo che non sia gia pieno altrimenti allarme

           FOR #i := "BTRK_LAYER_ITEMS" - 1 TO 1 BY -1 DO
               #ShiftArrayOk := MOVE_BLK_VARIANT(
                                                 SRC := "BTrk".A0303.Stacker.Layers[#i].Layer,
                                                 COUNT := 12,
                                                 SRC_INDEX := 0,
                                                 DEST_INDEX := 0,
                                                 DEST => "BTrk".A0303.Stacker.Layers[#i + 1].Layer);
           END_FOR;

           // Copia nuovo layer in Layers[1]
           // 
           IF #ShiftArrayOk = 0 THEN
               #TrkToStackerOk := MOVE_BLK_VARIANT(
                                                   SRC := "BTrk".A0303.Transfert.Layer,
                                                   COUNT := 12,
                                                   SRC_INDEX := 0,
                                                   DEST_INDEX := 0,
                                                   DEST => "BTrk".A0303.Stacker.Layers[1].Layer);

               IF #TrkToStackerOk = 0 THEN
                   "BTrk".A0303.Transfert.Layer := "BTrk".EmptyLayer;
               END_IF;

           END_IF;

       ELSE
           #Alarm.TrkStackerAlreadyFull := TRUE;
       END_IF;
   END_IF;
END_REGION

